LIN {X 0,Y 171.539,Z 336.57,A -85,B 0,C 180,E1 -22879.56,E2 -22879.56} C_VEL
LIN {X 0,Y 171.457,Z 336.598,A -85,B 0,C 180,E1 -22885.61,E2 -22885.61} C_VEL
LIN {X 0,Y 171.451,Z 336.623,A -85,B 0,C 180,E1 -22890.594,E2 -22890.594} C_VEL
LIN {X 0,Y 171.436,Z 336.681,A -85,B 0,C 180,E1 -22896.744,E2 -22896.744} C_VEL
LIN {X 0,Y 171.586,Z 337.511,A -85,B 0,C 180,E1 -22897.442,E2 -22897.442} C_VEL
LIN {X 0,Y 173.163,Z 340.46,A -85,B 0,C 180,E1 -22898.398,E2 -22898.398} C_VEL
LIN {X 0,Y 175.194,Z 342.365,A -85,B 0,C 180,E1 -22899.355,E2 -22899.355} C_VEL
LIN {X 0,Y 177.505,Z 345.855,A -85,B 0,C 180,E1 -22900.477,E2 -22900.477} C_VEL
LIN {X 0,Y 178.729,Z 347.281,A -85,B 0,C 180,E1 -22901.024,E2 -22901.024} C_VEL
LIN {X 0,Y 181.282,Z 350.846,A -85,B 0,C 180,E1 -22902.156,E2 -22902.156} C_VEL
LIN {X 0,Y 189.365,Z 363.13,A -85,B 0,C 180,E1 -22905.455,E2 -22905.455} C_VEL
LIN {X 0,Y 196.206,Z 374.838,A -85,B 0,C 180,E1 -22907.971,E2 -22907.971} C_VEL
LIN {X 0,Y 203.333,Z 389.329,A -85,B 0,C 180,E1 -22910.423,E2 -22910.423} C_VEL
LIN {X 0,Y 211.371,Z 406.535,A -85,B 0,C 180,E1 -22912.937,E2 -22912.937} C_VEL
LIN {X 0,Y 219.567,Z 420.322,A -85,B 0,C 180,E1 -22915.088,E2 -22915.088} C_VEL
LIN {X 0,Y 227.66,Z 431.79,A -85,B 0,C 180,E1 -22916.962,E2 -22916.962} C_VEL
LIN {X 0,Y 235.909,Z 442.056,A -85,B 0,C 180,E1 -22918.82,E2 -22918.82} C_VEL
LIN {X 0,Y 244.185,Z 451.427,A -85,B 0,C 180,E1 -22920.707,E2 -22920.707} C_VEL
LIN {X 0,Y 253.061,Z 460.521,A -85,B 0,C 180,E1 -22922.709,E2 -22922.709} C_VEL
LIN {X 0,Y 263.681,Z 469.922,A -85,B 0,C 180,E1 -22924.985,E2 -22924.985} C_VEL
LIN {X 0,Y 276.754,Z 479.974,A -85,B 0,C 180,E1 -22927.61,E2 -22927.61} C_VEL
LIN {X 0,Y 290.967,Z 490.138,A -85,B 0,C 180,E1 -22930.388,E2 -22930.388} C_VEL
LIN {X 0,Y 299.99,Z 496.755,A -85,B 0,C 180,E1 -22932.269,E2 -22932.269} C_VEL
LIN {X 0,Y 305.153,Z 500.286,A -85,B 0,C 180,E1 -22933.437,E2 -22933.437} C_VEL
LIN {X 0,Y 312.328,Z 505.427,A -85,B 0,C 180,E1 -22935.368,E2 -22935.368} C_VEL
LIN {X 0,Y 318.736,Z 509.419,A -85,B 0,C 180,E1 -22937.262,E2 -22937.262} C_VEL
LIN {X 0,Y 322.775,Z 512.115,A -85,B 0,C 180,E1 -22938.699,E2 -22938.699} C_VEL
LIN {X 0,Y 327.518,Z 515.418,A -85,B 0,C 180,E1 -22940.776,E2 -22940.776} C_VEL
LIN {X 0,Y 331.239,Z 517.603,A -85,B 0,C 180,E1 -22942.686,E2 -22942.686} C_VEL
LIN {X 0,Y 333.408,Z 518.666,A -85,B 0,C 180,E1 -22943.95,E2 -22943.95} C_VEL
LIN {X 0,Y 335.133,Z 519.458,A -85,B 0,C 180,E1 -22945.188,E2 -22945.188} C_VEL
LIN {X 0,Y 336.579,Z 519.977,A -85,B 0,C 180,E1 -22946.409,E2 -22946.409} C_VEL
LIN {X 0,Y 337.607,Z 520.419,A -85,B 0,C 180,E1 -22947.718,E2 -22947.718} C_VEL
LIN {X 0,Y 338.053,Z 520.65,A -85,B 0,C 180,E1 -22948.809,E2 -22948.809} C_VEL
LIN {X 0,Y 338.329,Z 520.665,A -85,B 0,C 180,E1 -22950,E2 -22950} C_VEL
LIN {X 0,Y 338.087,Z 520.616,A -85,B 0,C 180,E1 -22951.191,E2 -22951.191} C_VEL
LIN {X 0,Y 337.557,Z 520.347,A -85,B 0,C 180,E1 -22952.386,E2 -22952.386} C_VEL
LIN {X 0,Y 336.575,Z 519.955,A -85,B 0,C 180,E1 -22953.591,E2 -22953.591} C_VEL
LIN {X 0,Y 335.143,Z 519.423,A -85,B 0,C 180,E1 -22954.812,E2 -22954.812} C_VEL
LIN {X 0,Y 332.51,Z 518.272,A -85,B 0,C 180,E1 -22956.593,E2 -22956.593} C_VEL
LIN {X 0,Y 327.523,Z 515.378,A -85,B 0,C 180,E1 -22959.229,E2 -22959.229} C_VEL
LIN {X 0,Y 322.579,Z 512.01,A -85,B 0,C 180,E1 -22961.364,E2 -22961.364} C_VEL
LIN {X 0,Y 317.511,Z 508.69,A -85,B 0,C 180,E1 -22963.117,E2 -22963.117} C_VEL
LIN {X 0,Y 312.34,Z 505.397,A -85,B 0,C 180,E1 -22964.64,E2 -22964.64} C_VEL
LIN {X 0,Y 307.147,Z 501.743,A -85,B 0,C 180,E1 -22966.052,E2 -22966.052} C_VEL
LIN {X 0,Y 300.051,Z 496.781,A -85,B 0,C 180,E1 -22967.727,E2 -22967.727} C_VEL
LIN {X 0,Y 289.801,Z 489.324,A -85,B 0,C 180,E1 -22969.847,E2 -22969.847} C_VEL
LIN {X 0,Y 274.501,Z 478.341,A -85,B 0,C 180,E1 -22972.826,E2 -22972.826} C_VEL
LIN {X 0,Y 261.546,Z 468.134,A -85,B 0,C 180,E1 -22975.463,E2 -22975.463} C_VEL
LIN {X 0,Y 249.213,Z 456.773,A -85,B 0,C 180,E1 -22978.147,E2 -22978.147} C_VEL
LIN {X 0,Y 238.518,Z 445.13,A -85,B 0,C 180,E1 -22980.58,E2 -22980.58} C_VEL
LIN {X 0,Y 230.343,Z 435.166,A -85,B 0,C 180,E1 -22982.456,E2 -22982.456} C_VEL
LIN {X 0,Y 222.347,Z 424.476,A -85,B 0,C 180,E1 -22984.25,E2 -22984.25} C_VEL
LIN {X 0,Y 213.586,Z 410.542,A -85,B 0,C 180,E1 -22986.448,E2 -22986.448} C_VEL
LIN {X 0,Y 206.428,Z 396.381,A -85,B 0,C 180,E1 -22988.556,E2 -22988.556} C_VEL
LIN {X 0,Y 200.05,Z 382.426,A -85,B 0,C 180,E1 -22990.684,E2 -22990.684} C_VEL
LIN {X 0,Y 193.877,Z 370.717,A -85,B 0,C 180,E1 -22992.861,E2 -22992.861} C_VEL
LIN {X 0,Y 186.721,Z 358.92,A -85,B 0,C 180,E1 -22995.582,E2 -22995.582} C_VEL
LIN {X 0,Y 180.881,Z 350.422,A -85,B 0,C 180,E1 -22998.01,E2 -22998.01} C_VEL
LIN {X 0,Y 177.92,Z 346.242,A -85,B 0,C 180,E1 -22999.342,E2 -22999.342} C_VEL
LIN {X 0,Y 175.643,Z 343.253,A -85,B 0,C 180,E1 -23000.409,E2 -23000.409} C_VEL
LIN {X 0,Y 174.818,Z 341.844,A -85,B 0,C 180,E1 -23000.829,E2 -23000.829} C_VEL
LIN {X 0,Y 172.552,Z 339.652,A -85,B 0,C 180,E1 -23001.914,E2 -23001.914} C_VEL
LIN {X 0,Y 171.503,Z 337.185,A -85,B 0,C 180,E1 -23002.721,E2 -23002.721} C_VEL
LIN {X 0,Y 171.43,Z 336.639,A -85,B 0,C 180,E1 -23003.528,E2 -23003.528} C_VEL
LIN {X 0,Y 171.451,Z 336.623,A -85,B 0,C 180,E1 -23009.406,E2 -23009.406} C_VEL
LIN {X 0,Y 171.457,Z 336.598,A -85,B 0,C 180,E1 -23014.39,E2 -23014.39} C_VEL
LIN {X 0,Y 171.574,Z 336.565,A -85,B 0,C 180,E1 -23020.873,E2 -23020.873} C_VEL
LIN {X 0,Y 171.571,Z 336.612,A -85,B 0,C 180,E1 -23025.774,E2 -23025.774} C_VEL
LIN {X 0,Y 171.843,Z 336.526,A -85,B 0,C 180,E1 -23030.586,E2 -23030.586} C_VEL
LIN {X 0,Y 171.811,Z 336.582,A -85,B 0,C 180,E1 -23035.309,E2 -23035.309} C_VEL
LIN {X 0,Y 172.326,Z 336.463,A -85,B 0,C 180,E1 -23040.001,E2 -23040.001} C_VEL
LIN {X 0,Y 171.812,Z 336.584,A -85,B 0,C 180,E1 -23044.694,E2 -23044.694} C_VEL
LIN {X 0,Y 171.845,Z 336.523,A -85,B 0,C 180,E1 -23049.417,E2 -23049.417} C_VEL
LIN {X 0,Y 171.572,Z 336.611,A -85,B 0,C 180,E1 -23054.229,E2 -23054.229} C_VEL
LIN {X 0,Y 171.538,Z 336.57,A -85,B 0,C 180,E1 -23059.558,E2 -23059.558} C_VEL
LIN {X 0,Y 171.457,Z 336.59,A -85,B 0,C 180,E1 -23065.61,E2 -23065.61} C_VEL
LIN {X 0,Y 171.455,Z 336.629,A -85,B 0,C 180,E1 -23070.596,E2 -23070.596} C_VEL
LIN {X 0,Y 171.405,Z 336.708,A -85,B 0,C 180,E1 -23076.298,E2 -23076.298} C_VEL
LIN {X 0,Y 171.543,Z 337.483,A -85,B 0,C 180,E1 -23076.996,E2 -23076.996} C_VEL
LIN {X 0,Y 173.071,Z 340.36,A -85,B 0,C 180,E1 -23077.968,E2 -23077.968} C_VEL
LIN {X 0,Y 175.48,Z 343.334,A -85,B 0,C 180,E1 -23079.147,E2 -23079.147} C_VEL
LIN {X 0,Y 178.282,Z 347.76,A -85,B 0,C 180,E1 -23080.502,E2 -23080.502} C_VEL
LIN {X 0,Y 182.818,Z 355.351,A -85,B 0,C 180,E1 -23082.561,E2 -23082.561} C_VEL
LIN {X 0,Y 189.402,Z 367.454,A -85,B 0,C 180,E1 -23085.307,E2 -23085.307} C_VEL
LIN {X 0,Y 194.801,Z 378.934,A -85,B 0,C 180,E1 -23087.411,E2 -23087.411} C_VEL
LIN {X 0,Y 199.89,Z 391.574,A -85,B 0,C 180,E1 -23089.317,E2 -23089.317} C_VEL
LIN {X 0,Y 201.451,Z 403.372,A -85,B 0,C 180,E1 -23090.231,E2 -23090.231} C_VEL
LIN {X 0,Y 199.159,Z 444.488,A -85,B 0,C 180,E1 -23091.639,E2 -23091.639} C_VEL
LIN {X 0,Y 197.867,Z 455.855,A -85,B 0,C 180,E1 -23092.266,E2 -23092.266} C_VEL
LIN {X 0,Y 195.589,Z 468.974,A -85,B 0,C 180,E1 -23093.319,E2 -23093.319} C_VEL
LIN {X 0,Y 192.896,Z 480.518,A -85,B 0,C 180,E1 -23094.663,E2 -23094.663} C_VEL
LIN {X 0,Y 190.383,Z 489.79,A -85,B 0,C 180,E1 -23096.06,E2 -23096.06} C_VEL
LIN {X 0,Y 187.56,Z 498.728,A -85,B 0,C 180,E1 -23097.728,E2 -23097.728} C_VEL
LIN {X 0,Y 184.613,Z 507.253,A -85,B 0,C 180,E1 -23099.709,E2 -23099.709} C_VEL
LIN {X 0,Y 181.877,Z 514.468,A -85,B 0,C 180,E1 -23101.748,E2 -23101.748} C_VEL
LIN {X 0,Y 179.451,Z 520.668,A -85,B 0,C 180,E1 -23103.859,E2 -23103.859} C_VEL
LIN {X 0,Y 176.902,Z 527.209,A -85,B 0,C 180,E1 -23106.592,E2 -23106.592} C_VEL
LIN {X 0,Y 174.939,Z 531.708,A -85,B 0,C 180,E1 -23108.804,E2 -23108.804} C_VEL
LIN {X 0,Y 172.581,Z 537.2,A -85,B 0,C 180,E1 -23112.217,E2 -23112.217} C_VEL
LIN {X 0,Y 170.823,Z 541.528,A -85,B 0,C 180,E1 -23115.709,E2 -23115.709} C_VEL
LIN {X 0,Y 170.023,Z 543.9,A -85,B 0,C 180,E1 -23118.073,E2 -23118.073} C_VEL
LIN {X 0,Y 169.422,Z 545.703,A -85,B 0,C 180,E1 -23120.449,E2 -23120.449} C_VEL
LIN {X 0,Y 168.933,Z 548.162,A -85,B 0,C 180,E1 -23125.227,E2 -23125.227} C_VEL
LIN {X 0,Y 168.87,Z 548.808,A -85,B 0,C 180,E1 -23128.406,E2 -23128.406} C_VEL
LIN {X 0,Y 168.968,Z 548.914,A -85,B 0,C 180,E1 -23130,E2 -23130} C_VEL
LIN {X 0,Y 168.853,Z 548.695,A -85,B 0,C 180,E1 -23132.627,E2 -23132.627} C_VEL
LIN {X 0,Y 168.866,Z 548.16,A -85,B 0,C 180,E1 -23134.775,E2 -23134.775} C_VEL
LIN {X 0,Y 169.235,Z 546.252,A -85,B 0,C 180,E1 -23138.613,E2 -23138.613} C_VEL
LIN {X 0,Y 168.968,Z 544.98,A -85,B 0,C 180,E1 -23140.565,E2 -23140.565} C_VEL
LIN {X 0,Y 167.056,Z 542.347,A -85,B 0,C 180,E1 -23143.761,E2 -23143.761} C_VEL
LIN {X 0,Y 165.58,Z 539.031,A -85,B 0,C 180,E1 -23146.945,E2 -23146.945} C_VEL
LIN {X 0,Y 165.998,Z 536.621,A -85,B 0,C 180,E1 -23148.811,E2 -23148.811} C_VEL
LIN {X 0,Y 168.812,Z 530.478,A -85,B 0,C 180,E1 -23152.649,E2 -23152.649} C_VEL
LIN {X 0,Y 171.522,Z 524.246,A -85,B 0,C 180,E1 -23155.65,E2 -23155.65} C_VEL
LIN {X 0,Y 174.325,Z 517.526,A -85,B 0,C 180,E1 -23158.274,E2 -23158.274} C_VEL
LIN {X 0,Y 177.771,Z 508.977,A -85,B 0,C 180,E1 -23160.926,E2 -23160.926} C_VEL
LIN {X 0,Y 180.808,Z 500.803,A -85,B 0,C 180,E1 -23162.968,E2 -23162.968} C_VEL
LIN {X 0,Y 183.669,Z 492.297,A -85,B 0,C 180,E1 -23164.692,E2 -23164.692} C_VEL
LIN {X 0,Y 186.244,Z 483.585,A -85,B 0,C 180,E1 -23166.129,E2 -23166.129} C_VEL
LIN {X 0,Y 188.762,Z 473.833,A -85,B 0,C 180,E1 -23167.397,E2 -23167.397} C_VEL
LIN {X 0,Y 190.897,Z 463.758,A -85,B 0,C 180,E1 -23168.407,E2 -23168.407} C_VEL
LIN {X 0,Y 192.63,Z 453.291,A -85,B 0,C 180,E1 -23169.178,E2 -23169.178} C_VEL
LIN {X 0,Y 193.719,Z 443.215,A -85,B 0,C 180,E1 -23169.709,E2 -23169.709} C_VEL
LIN {X 0,Y 195.93,Z 403.202,A -85,B 0,C 180,E1 -23171.124,E2 -23171.124} C_VEL
LIN {X 0,Y 194.544,Z 393.897,A -85,B 0,C 180,E1 -23171.929,E2 -23171.929} C_VEL
LIN {X 0,Y 189.257,Z 380.763,A -85,B 0,C 180,E1 -23174.046,E2 -23174.046} C_VEL
LIN {X 0,Y 184.606,Z 370.872,A -85,B 0,C 180,E1 -23175.988,E2 -23175.988} C_VEL
LIN {X 0,Y 177.81,Z 358.124,A -85,B 0,C 180,E1 -23179.048,E2 -23179.048} C_VEL
LIN {X 0,Y 173.971,Z 351.983,A -85,B 0,C 180,E1 -23180.907,E2 -23180.907} C_VEL
LIN {X 0,Y 171.184,Z 347.548,A -85,B 0,C 180,E1 -23182.358,E2 -23182.358} C_VEL
LIN {X 0,Y 168.609,Z 344.054,A -85,B 0,C 180,E1 -23183.744,E2 -23183.744} C_VEL
LIN {X 0,Y 167.778,Z 342.747,A -85,B 0,C 180,E1 -23184.224,E2 -23184.224} C_VEL
LIN {X 0,Y 165.411,Z 340.457,A -85,B 0,C 180,E1 -23185.54,E2 -23185.54} C_VEL
LIN {X 0,Y 164.431,Z 338.113,A -85,B 0,C 180,E1 -23186.418,E2 -23186.418} C_VEL
LIN {X 0,Y 164.369,Z 337.528,A -85,B 0,C 180,E1 -23187.272,E2 -23187.272} C_VEL
LIN {X 0,Y 164.337,Z 337.477,A -85,B 0,C 180,E1 -23191.937,E2 -23191.937} C_VEL
LIN {X 0,Y 164.405,Z 337.47,A -85,B 0,C 180,E1 -23194.691,E2 -23194.691} C_VEL
LIN {X 0,Y 164.483,Z 337.45,A -85,B 0,C 180,E1 -23200.05,E2 -23200.05} C_VEL
LIN {X 0,Y 164.52,Z 337.482,A -85,B 0,C 180,E1 -23205.147,E2 -23205.147} C_VEL
LIN {X 0,Y 164.765,Z 337.405,A -85,B 0,C 180,E1 -23210.175,E2 -23210.175} C_VEL
LIN {X 0,Y 164.827,Z 337.411,A -85,B 0,C 180,E1 -23212.649,E2 -23212.649} C_VEL
LIN {X 0,Y 165.044,Z 337.393,A -85,B 0,C 180,E1 -23217.558,E2 -23217.558} C_VEL
LIN {X 0,Y 165.289,Z 337.339,A -85,B 0,C 180,E1 -23219.999,E2 -23219.999} C_VEL
LIN {X 0,Y 164.76,Z 337.461,A -85,B 0,C 180,E1 -23224.893,E2 -23224.893} C_VEL
LIN {X 0,Y 164.826,Z 337.421,A -85,B 0,C 180,E1 -23227.348,E2 -23227.348} C_VEL
LIN {X 0,Y 164.699,Z 337.418,A -85,B 0,C 180,E1 -23231.059,E2 -23231.059} C_VEL
LIN {X 0,Y 164.519,Z 337.493,A -85,B 0,C 180,E1 -23234.85,E2 -23234.85} C_VEL
LIN {X 0,Y 164.469,Z 337.452,A -85,B 0,C 180,E1 -23239.988,E2 -23239.988} C_VEL
LIN {X 0,Y 164.383,Z 337.474,A -85,B 0,C 180,E1 -23246.129,E2 -23246.129} C_VEL
LIN {X 0,Y 164.383,Z 337.492,A -85,B 0,C 180,E1 -23252.377,E2 -23252.377} C_VEL
LIN {X 0,Y 164.374,Z 337.825,A -85,B 0,C 180,E1 -23253.766,E2 -23253.766} C_VEL
LIN {X 0,Y 164.716,Z 339.072,A -85,B 0,C 180,E1 -23254.365,E2 -23254.365} C_VEL
LIN {X 0,Y 166.42,Z 341.678,A -85,B 0,C 180,E1 -23255.433,E2 -23255.433} C_VEL
LIN {X 0,Y 168.28,Z 343.196,A -85,B 0,C 180,E1 -23256.427,E2 -23256.427} C_VEL
LIN {X 0,Y 170.447,Z 346.622,A -85,B 0,C 180,E1 -23257.643,E2 -23257.643} C_VEL
LIN {X 0,Y 172.181,Z 348.499,A -85,B 0,C 180,E1 -23258.514,E2 -23258.514} C_VEL
LIN {X 0,Y 174.855,Z 352.169,A -85,B 0,C 180,E1 -23259.841,E2 -23259.841} C_VEL
LIN {X 0,Y 181.754,Z 362.408,A -85,B 0,C 180,E1 -23262.984,E2 -23262.984} C_VEL
LIN {X 0,Y 187.458,Z 371.661,A -85,B 0,C 180,E1 -23265.327,E2 -23265.327} C_VEL
LIN {X 0,Y 192.641,Z 380.983,A -85,B 0,C 180,E1 -23267.308,E2 -23267.308} C_VEL
LIN {X 0,Y 198.981,Z 394.263,A -85,B 0,C 180,E1 -23269.602,E2 -23269.602} C_VEL
LIN {X 0,Y 206.603,Z 410.847,A -85,B 0,C 180,E1 -23272.111,E2 -23272.111} C_VEL
LIN {X 0,Y 214.984,Z 425.115,A -85,B 0,C 180,E1 -23274.419,E2 -23274.419} C_VEL
LIN {X 0,Y 222.86,Z 436.51,A -85,B 0,C 180,E1 -23276.379,E2 -23276.379} C_VEL
LIN {X 0,Y 232.034,Z 448.156,A -85,B 0,C 180,E1 -23278.684,E2 -23278.684} C_VEL
LIN {X 0,Y 241.126,Z 458.487,A -85,B 0,C 180,E1 -23280.971,E2 -23280.971} C_VEL
LIN {X 0,Y 250.242,Z 467.531,A -85,B 0,C 180,E1 -23283.174,E2 -23283.174} C_VEL
LIN {X 0,Y 261.923,Z 477.462,A -85,B 0,C 180,E1 -23285.823,E2 -23285.823} C_VEL
LIN {X 0,Y 276.505,Z 488.237,A -85,B 0,C 180,E1 -23288.897,E2 -23288.897} C_VEL
LIN {X 0,Y 289.062,Z 496.933,A -85,B 0,C 180,E1 -23291.477,E2 -23291.477} C_VEL
LIN {X 0,Y 298.844,Z 503.742,A -85,B 0,C 180,E1 -23293.608,E2 -23293.608} C_VEL
LIN {X 0,Y 305.422,Z 508.49,A -85,B 0,C 180,E1 -23295.338,E2 -23295.338} C_VEL
LIN {X 0,Y 311.013,Z 512.125,A -85,B 0,C 180,E1 -23296.94,E2 -23296.94} C_VEL
LIN {X 0,Y 315.674,Z 515.006,A -85,B 0,C 180,E1 -23298.442,E2 -23298.442} C_VEL
LIN {X 0,Y 320.633,Z 518.493,A -85,B 0,C 180,E1 -23300.521,E2 -23300.521} C_VEL
LIN {X 0,Y 325.665,Z 521.536,A -85,B 0,C 180,E1 -23303.066,E2 -23303.066} C_VEL
LIN {X 0,Y 328.836,Z 523.081,A -85,B 0,C 180,E1 -23305.096,E2 -23305.096} C_VEL
LIN {X 0,Y 330.825,Z 523.835,A -85,B 0,C 180,E1 -23306.805,E2 -23306.805} C_VEL
LIN {X 0,Y 331.972,Z 524.341,A -85,B 0,C 180,E1 -23308.787,E2 -23308.787} C_VEL
LIN {X 0,Y 332.28,Z 524.36,A -85,B 0,C 180,E1 -23310,E2 -23310} C_VEL
LIN {X 0,Y 332.008,Z 524.312,A -85,B 0,C 180,E1 -23311.213,E2 -23311.213} C_VEL
LIN {X 0,Y 330.826,Z 523.842,A -85,B 0,C 180,E1 -23313.198,E2 -23313.198} C_VEL
LIN {X 0,Y 328.857,Z 523.049,A -85,B 0,C 180,E1 -23314.904,E2 -23314.904} C_VEL
LIN {X 0,Y 325.667,Z 521.523,A -85,B 0,C 180,E1 -23316.937,E2 -23316.937} C_VEL
LIN {X 0,Y 322.114,Z 519.453,A -85,B 0,C 180,E1 -23318.785,E2 -23318.785} C_VEL
LIN {X 0,Y 319.122,Z 517.476,A -85,B 0,C 180,E1 -23320.147,E2 -23320.147} C_VEL
LIN {X 0,Y 315.636,Z 515.014,A -85,B 0,C 180,E1 -23321.566,E2 -23321.566} C_VEL
LIN {X 0,Y 310.45,Z 511.729,A -85,B 0,C 180,E1 -23323.239,E2 -23323.239} C_VEL
LIN {X 0,Y 305.201,Z 508.34,A -85,B 0,C 180,E1 -23324.729,E2 -23324.729} C_VEL
LIN {X 0,Y 298.749,Z 503.734,A -85,B 0,C 180,E1 -23326.397,E2 -23326.397} C_VEL
LIN {X 0,Y 291.782,Z 498.874,A -85,B 0,C 180,E1 -23327.939,E2 -23327.939} C_VEL
LIN {X 0,Y 283.585,Z 493.015,A -85,B 0,C 180,E1 -23329.656,E2 -23329.656} C_VEL
LIN {X 0,Y 272.673,Z 485.406,A -85,B 0,C 180,E1 -23331.896,E2 -23331.896} C_VEL
LIN {X 0,Y 261.917,Z 477.484,A -85,B 0,C 180,E1 -23334.175,E2 -23334.175} C_VEL
LIN {X 0,Y 250.239,Z 467.543,A -85,B 0,C 180,E1 -23336.824,E2 -23336.824} C_VEL
LIN {X 0,Y 241.128,Z 458.477,A -85,B 0,C 180,E1 -23339.029,E2 -23339.029} C_VEL
LIN {X 0,Y 230.977,Z 446.931,A -85,B 0,C 180,E1 -23341.576,E2 -23341.576} C_VEL
LIN {X 0,Y 221.582,Z 434.806,A -85,B 0,C 180,E1 -23343.944,E2 -23343.944} C_VEL
LIN {X 0,Y 211.908,Z 420.264,A -85,B 0,C 180,E1 -23346.383,E2 -23346.383} C_VEL
LIN {X 0,Y 204.622,Z 406.869,A -85,B 0,C 180,E1 -23348.5,E2 -23348.5} C_VEL
LIN {X 0,Y 195.301,Z 386.39,A -85,B 0,C 180,E1 -23351.709,E2 -23351.709} C_VEL
LIN {X 0,Y 189.403,Z 374.942,A -85,B 0,C 180,E1 -23353.92,E2 -23353.92} C_VEL
LIN {X 0,Y 182.781,Z 363.899,A -85,B 0,C 180,E1 -23356.585,E2 -23356.585} C_VEL
LIN {X 0,Y 176.957,Z 355.329,A -85,B 0,C 180,E1 -23359.151,E2 -23359.151} C_VEL
LIN {X 0,Y 174.25,Z 351.474,A -85,B 0,C 180,E1 -23360.444,E2 -23360.444} C_VEL
LIN {X 0,Y 171.46,Z 347.586,A -85,B 0,C 180,E1 -23361.853,E2 -23361.853} C_VEL
LIN {X 0,Y 169.045,Z 344.703,A -85,B 0,C 180,E1 -23363.115,E2 -23363.115} C_VEL
LIN {X 0,Y 167.929,Z 342.817,A -85,B 0,C 180,E1 -23363.763,E2 -23363.763} C_VEL
LIN {X 0,Y 165.707,Z 340.823,A -85,B 0,C 180,E1 -23364.981,E2 -23364.981} C_VEL
LIN {X 0,Y 164.437,Z 338.037,A -85,B 0,C 180,E1 -23366.04,E2 -23366.04} C_VEL
LIN {X 0,Y 164.342,Z 337.513,A -85,B 0,C 180,E1 -23366.923,E2 -23366.923} C_VEL
LIN {X 0,Y 164.398,Z 337.505,A -85,B 0,C 180,E1 -23369.138,E2 -23369.138} C_VEL
LIN {X 0,Y 164.405,Z 337.479,A -85,B 0,C 180,E1 -23374.694,E2 -23374.694} C_VEL
LIN {X 0,Y 164.481,Z 337.45,A -85,B 0,C 180,E1 -23380.052,E2 -23380.052} C_VEL
LIN {X 0,Y 164.519,Z 337.493,A -85,B 0,C 180,E1 -23385.15,E2 -23385.15} C_VEL
LIN {X 0,Y 164.763,Z 337.407,A -85,B 0,C 180,E1 -23390.178,E2 -23390.178} C_VEL
LIN {X 0,Y 164.826,Z 337.421,A -85,B 0,C 180,E1 -23392.652,E2 -23392.652} C_VEL
LIN {X 0,Y 165.043,Z 337.383,A -85,B 0,C 180,E1 -23397.561,E2 -23397.561} C_VEL
LIN {X 0,Y 165.289,Z 337.339,A -85,B 0,C 180,E1 -23400.001,E2 -23400.001} C_VEL
LIN {X 0,Y 164.761,Z 337.461,A -85,B 0,C 180,E1 -23404.895,E2 -23404.895} C_VEL
LIN {X 0,Y 164.827,Z 337.411,A -85,B 0,C 180,E1 -23407.351,E2 -23407.351} C_VEL
LIN {X 0,Y 164.7,Z 337.42,A -85,B 0,C 180,E1 -23411.062,E2 -23411.062} C_VEL
LIN {X 0,Y 164.478,Z 337.449,A -85,B 0,C 180,E1 -23417.405,E2 -23417.405} C_VEL
LIN {X 0,Y 164.471,Z 337.452,A -85,B 0,C 180,E1 -23419.991,E2 -23419.991} C_VEL
LIN {X 0,Y 164.384,Z 337.468,A -85,B 0,C 180,E1 -23426.129,E2 -23426.129} C_VEL
LIN {X 0,Y 164.385,Z 337.5,A -85,B 0,C 180,E1 -23432.38,E2 -23432.38} C_VEL
LIN {X 0,Y 164.408,Z 337.879,A -85,B 0,C 180,E1 -23433.413,E2 -23433.413} C_VEL
LIN {X 0,Y 164.788,Z 339.234,A -85,B 0,C 180,E1 -23434.036,E2 -23434.036} C_VEL
LIN {X 0,Y 166.493,Z 341.748,A -85,B 0,C 180,E1 -23435.089,E2 -23435.089} C_VEL
LIN {X 0,Y 168.296,Z 343.276,A -85,B 0,C 180,E1 -23436.056,E2 -23436.056} C_VEL
LIN {X 0,Y 170.346,Z 346.513,A -85,B 0,C 180,E1 -23437.207,E2 -23437.207} C_VEL
LIN {X 0,Y 172.227,Z 349.051,A -85,B 0,C 180,E1 -23438.185,E2 -23438.185} C_VEL
LIN {X 0,Y 176.235,Z 355.622,A -85,B 0,C 180,E1 -23440.209,E2 -23440.209} C_VEL
LIN {X 0,Y 180.315,Z 362.639,A -85,B 0,C 180,E1 -23442.117,E2 -23442.117} C_VEL
LIN {X 0,Y 187.188,Z 376.123,A -85,B 0,C 180,E1 -23445.097,E2 -23445.097} C_VEL
LIN {X 0,Y 192.937,Z 389.661,A -85,B 0,C 180,E1 -23447.435,E2 -23447.435} C_VEL
LIN {X 0,Y 194.8,Z 394.774,A -85,B 0,C 180,E1 -23448.181,E2 -23448.181} C_VEL
LIN {X 0,Y 195.977,Z 403.646,A -85,B 0,C 180,E1 -23448.909,E2 -23448.909} C_VEL
LIN {X 0,Y 193.648,Z 444.156,A -85,B 0,C 180,E1 -23450.327,E2 -23450.327} C_VEL
LIN {X 0,Y 192.398,Z 454.945,A -85,B 0,C 180,E1 -23450.925,E2 -23450.925} C_VEL
LIN {X 0,Y 190.447,Z 466.333,A -85,B 0,C 180,E1 -23451.822,E2 -23451.822} C_VEL
LIN {X 0,Y 187.641,Z 478.692,A -85,B 0,C 180,E1 -23453.183,E2 -23453.183} C_VEL
LIN {X 0,Y 184.536,Z 489.596,A -85,B 0,C 180,E1 -23454.829,E2 -23454.829} C_VEL
LIN {X 0,Y 181.597,Z 498.534,A -85,B 0,C 180,E1 -23456.532,E2 -23456.532} C_VEL
LIN {X 0,Y 178.487,Z 507.058,A -85,B 0,C 180,E1 -23458.553,E2 -23458.553} C_VEL
LIN {X 0,Y 175.632,Z 514.273,A -85,B 0,C 180,E1 -23460.648,E2 -23460.648} C_VEL
LIN {X 0,Y 173.076,Z 520.473,A -85,B 0,C 180,E1 -23462.818,E2 -23462.818} C_VEL
LIN {X 0,Y 170.38,Z 527.014,A -85,B 0,C 180,E1 -23465.639,E2 -23465.639} C_VEL
LIN {X 0,Y 168.309,Z 531.513,A -85,B 0,C 180,E1 -23467.926,E2 -23467.926} C_VEL
LIN {X 0,Y 165.822,Z 537.006,A -85,B 0,C 180,E1 -23471.466,E2 -23471.466} C_VEL
LIN {X 0,Y 163.901,Z 541.333,A -85,B 0,C 180,E1 -23475.092,E2 -23475.092} C_VEL
LIN {X 0,Y 163.054,Z 543.705,A -85,B 0,C 180,E1 -23477.555,E2 -23477.555} C_VEL
LIN {X 0,Y 162.403,Z 545.509,A -85,B 0,C 180,E1 -23480.032,E2 -23480.032} C_VEL
LIN {X 0,Y 161.852,Z 547.968,A -85,B 0,C 180,E1 -23485.018,E2 -23485.018} C_VEL
LIN {X 0,Y 161.8,Z 548.562,A -85,B 0,C 180,E1 -23487.511,E2 -23487.511} C_VEL
LIN {X 0,Y 161.884,Z 548.721,A -85,B 0,C 180,E1 -23490,E2 -23490} C_VEL
LIN {X 0,Y 161.763,Z 548.561,A -85,B 0,C 180,E1 -23492.49,E2 -23492.49} C_VEL
LIN {X 0,Y 161.771,Z 547.966,A -85,B 0,C 180,E1 -23494.984,E2 -23494.984} C_VEL
LIN {X 0,Y 162.4,Z 545.509,A -85,B 0,C 180,E1 -23499.968,E2 -23499.968} C_VEL
LIN {X 0,Y 163.453,Z 542.552,A -85,B 0,C 180,E1 -23503.679,E2 -23503.679} C_VEL
LIN {X 0,Y 165.066,Z 538.559,A -85,B 0,C 180,E1 -23507.339,E2 -23507.339} C_VEL
LIN {X 0,Y 165.998,Z 536.621,A -85,B 0,C 180,E1 -23508.811,E2 -23508.811} C_VEL
LIN {X 0,Y 166.559,Z 534.024,A -85,B 0,C 180,E1 -23510.629,E2 -23510.629} C_VEL
LIN {X 0,Y 165.964,Z 529.362,A -85,B 0,C 180,E1 -23513.643,E2 -23513.643} C_VEL
LIN {X 0,Y 165.65,Z 524.205,A -85,B 0,C 180,E1 -23516.563,E2 -23516.563} C_VEL
LIN {X 0,Y 166.625,Z 520.588,A -85,B 0,C 180,E1 -23518.173,E2 -23518.173} C_VEL
LIN {X 0,Y 170.198,Z 512.453,A -85,B 0,C 180,E1 -23521.074,E2 -23521.074} C_VEL
LIN {X 0,Y 174.459,Z 501.742,A -85,B 0,C 180,E1 -23523.982,E2 -23523.982} C_VEL
LIN {X 0,Y 177.461,Z 493.455,A -85,B 0,C 180,E1 -23525.742,E2 -23525.742} C_VEL
LIN {X 0,Y 180.554,Z 483.391,A -85,B 0,C 180,E1 -23527.458,E2 -23527.458} C_VEL
LIN {X 0,Y 183.181,Z 473.64,A -85,B 0,C 180,E1 -23528.744,E2 -23528.744} C_VEL
LIN {X 0,Y 185.391,Z 463.564,A -85,B 0,C 180,E1 -23529.769,E2 -23529.769} C_VEL
LIN {X 0,Y 187.175,Z 453.147,A -85,B 0,C 180,E1 -23530.547,E2 -23530.547} C_VEL
LIN {X 0,Y 188.292,Z 443.238,A -85,B 0,C 180,E1 -23531.08,E2 -23531.08} C_VEL
LIN {X 0,Y 190.573,Z 404.451,A -85,B 0,C 180,E1 -23532.474,E2 -23532.474} C_VEL
LIN {X 0,Y 189.457,Z 396.777,A -85,B 0,C 180,E1 -23533.17,E2 -23533.17} C_VEL
LIN {X 0,Y 184.427,Z 384.044,A -85,B 0,C 180,E1 -23535.328,E2 -23535.328} C_VEL
LIN {X 0,Y 180.286,Z 375.137,A -85,B 0,C 180,E1 -23537.173,E2 -23537.173} C_VEL
LIN {X 0,Y 174.016,Z 363.082,A -85,B 0,C 180,E1 -23540.186,E2 -23540.186} C_VEL
LIN {X 0,Y 170.397,Z 357.048,A -85,B 0,C 180,E1 -23542.061,E2 -23542.061} C_VEL
LIN {X 0,Y 167.74,Z 352.846,A -85,B 0,C 180,E1 -23543.526,E2 -23543.526} C_VEL
LIN {X 0,Y 164.723,Z 348.661,A -85,B 0,C 180,E1 -23545.271,E2 -23545.271} C_VEL
LIN {X 0,Y 162.165,Z 345.621,A -85,B 0,C 180,E1 -23546.827,E2 -23546.827} C_VEL
LIN {X 0,Y 161.152,Z 343.832,A -85,B 0,C 180,E1 -23547.522,E2 -23547.522} C_VEL
LIN {X 0,Y 158.719,Z 341.761,A -85,B 0,C 180,E1 -23549.095,E2 -23549.095} C_VEL
LIN {X 0,Y 157.402,Z 338.94,A -85,B 0,C 180,E1 -23550.399,E2 -23550.399} C_VEL
LIN {X 0,Y 157.293,Z 338.412,A -85,B 0,C 180,E1 -23551.293,E2 -23551.293} C_VEL
LIN {X 0,Y 157.302,Z 338.376,A -85,B 0,C 180,E1 -23556.289,E2 -23556.289} C_VEL
LIN {X 0,Y 157.406,Z 338.325,A -85,B 0,C 180,E1 -23561.786,E2 -23561.786} C_VEL
LIN {X 0,Y 157.526,Z 338.34,A -85,B 0,C 180,E1 -23567.109,E2 -23567.109} C_VEL
LIN {X 0,Y 157.686,Z 338.287,A -85,B 0,C 180,E1 -23569.729,E2 -23569.729} C_VEL
LIN {X 0,Y 157.764,Z 338.285,A -85,B 0,C 180,E1 -23572.318,E2 -23572.318} C_VEL
LIN {X 0,Y 158.252,Z 338.215,A -85,B 0,C 180,E1 -23579.999,E2 -23579.999} C_VEL
LIN {X 0,Y 157.763,Z 338.294,A -85,B 0,C 180,E1 -23587.679,E2 -23587.679} C_VEL
LIN {X 0,Y 157.63,Z 338.299,A -85,B 0,C 180,E1 -23591.229,E2 -23591.229} C_VEL
LIN {X 0,Y 157.449,Z 338.363,A -85,B 0,C 180,E1 -23595.533,E2 -23595.533} C_VEL
LIN {X 0,Y 157.365,Z 338.343,A -85,B 0,C 180,E1 -23600.932,E2 -23600.932} C_VEL
LIN {X 0,Y 157.305,Z 338.351,A -85,B 0,C 180,E1 -23606.68,E2 -23606.68} C_VEL
LIN {X 0,Y 157.336,Z 338.675,A -85,B 0,C 180,E1 -23609.704,E2 -23609.704} C_VEL
LIN {X 0,Y 157.686,Z 339.847,A -85,B 0,C 180,E1 -23610.461,E2 -23610.461} C_VEL
LIN {X 0,Y 159.21,Z 342.375,A -85,B 0,C 180,E1 -23611.633,E2 -23611.633} C_VEL
LIN {X 0,Y 161.456,Z 344.136,A -85,B 0,C 180,E1 -23613.055,E2 -23613.055} C_VEL
LIN {X 0,Y 163.488,Z 347.447,A -85,B 0,C 180,E1 -23614.395,E2 -23614.395} C_VEL
LIN {X 0,Y 165.523,Z 349.552,A -85,B 0,C 180,E1 -23615.573,E2 -23615.573} C_VEL
LIN {X 0,Y 168.088,Z 353.12,A -85,B 0,C 180,E1 -23617.036,E2 -23617.036} C_VEL
LIN {X 0,Y 169.381,Z 354.84,A -85,B 0,C 180,E1 -23617.733,E2 -23617.733} C_VEL
LIN {X 0,Y 172.835,Z 359.785,A -85,B 0,C 180,E1 -23619.518,E2 -23619.518} C_VEL
LIN {X 0,Y 177.448,Z 366.628,A -85,B 0,C 180,E1 -23621.713,E2 -23621.713} C_VEL
LIN {X 0,Y 183.213,Z 376.139,A -85,B 0,C 180,E1 -23624.238,E2 -23624.238} C_VEL
LIN {X 0,Y 188.806,Z 386.509,A -85,B 0,C 180,E1 -23626.503,E2 -23626.503} C_VEL
LIN {X 0,Y 194.884,Z 399.727,A -85,B 0,C 180,E1 -23628.826,E2 -23628.826} C_VEL
LIN {X 0,Y 201.868,Z 415.137,A -85,B 0,C 180,E1 -23631.243,E2 -23631.243} C_VEL
LIN {X 0,Y 210.208,Z 429.561,A -85,B 0,C 180,E1 -23633.66,E2 -23633.66} C_VEL
LIN {X 0,Y 217.978,Z 441.2,A -85,B 0,C 180,E1 -23635.811,E2 -23635.811} C_VEL
LIN {X 0,Y 226.168,Z 451.966,A -85,B 0,C 180,E1 -23638.113,E2 -23638.113} C_VEL
LIN {X 0,Y 235.644,Z 462.961,A -85,B 0,C 180,E1 -23640.733,E2 -23640.733} C_VEL
LIN {X 0,Y 244.421,Z 471.804,A -85,B 0,C 180,E1 -23643.043,E2 -23643.043} C_VEL
LIN {X 0,Y 254.732,Z 480.684,A -85,B 0,C 180,E1 -23645.567,E2 -23645.567} C_VEL
LIN {X 0,Y 269.065,Z 491.142,A -85,B 0,C 180,E1 -23648.784,E2 -23648.784} C_VEL
LIN {X 0,Y 281.649,Z 499.573,A -85,B 0,C 180,E1 -23651.478,E2 -23651.478} C_VEL
LIN {X 0,Y 292.58,Z 506.972,A -85,B 0,C 180,E1 -23653.907,E2 -23653.907} C_VEL
LIN {X 0,Y 299.526,Z 511.961,A -85,B 0,C 180,E1 -23655.705,E2 -23655.705} C_VEL
LIN {X 0,Y 304.711,Z 515.359,A -85,B 0,C 180,E1 -23657.169,E2 -23657.169} C_VEL
LIN {X 0,Y 309.779,Z 518.479,A -85,B 0,C 180,E1 -23658.776,E2 -23658.776} C_VEL
LIN {X 0,Y 313.638,Z 521.233,A -85,B 0,C 180,E1 -23660.38,E2 -23660.38} C_VEL
LIN {X 0,Y 318.729,Z 524.435,A -85,B 0,C 180,E1 -23662.857,E2 -23662.857} C_VEL
LIN {X 0,Y 322.203,Z 526.16,A -85,B 0,C 180,E1 -23664.995,E2 -23664.995} C_VEL
LIN {X 0,Y 323.942,Z 526.888,A -85,B 0,C 180,E1 -23666.345,E2 -23666.345} C_VEL
LIN {X 0,Y 325.024,Z 527.31,A -85,B 0,C 180,E1 -23667.521,E2 -23667.521} C_VEL
LIN {X 0,Y 325.649,Z 527.595,A -85,B 0,C 180,E1 -23668.763,E2 -23668.763} C_VEL
LIN {X 0,Y 325.969,Z 527.628,A -85,B 0,C 180,E1 -23670,E2 -23670} C_VEL
LIN {X 0,Y 325.678,Z 527.574,A -85,B 0,C 180,E1 -23671.236,E2 -23671.236} C_VEL
LIN {X 0,Y 325.06,Z 527.283,A -85,B 0,C 180,E1 -23672.478,E2 -23672.478} C_VEL
LIN {X 0,Y 323.852,Z 526.836,A -85,B 0,C 180,E1 -23673.733,E2 -23673.733} C_VEL
LIN {X 0,Y 322.21,Z 526.152,A -85,B 0,C 180,E1 -23675.005,E2 -23675.005} C_VEL
LIN {X 0,Y 318.726,Z 524.412,A -85,B 0,C 180,E1 -23677.139,E2 -23677.139} C_VEL
LIN {X 0,Y 315.043,Z 522.188,A -85,B 0,C 180,E1 -23678.984,E2 -23678.984} C_VEL
LIN {X 0,Y 311.837,Z 519.993,A -85,B 0,C 180,E1 -23680.387,E2 -23680.387} C_VEL
LIN {X 0,Y 307.879,Z 517.302,A -85,B 0,C 180,E1 -23681.855,E2 -23681.855} C_VEL
LIN {X 0,Y 302.663,Z 514.008,A -85,B 0,C 180,E1 -23683.427,E2 -23683.427} C_VEL
LIN {X 0,Y 296.485,Z 509.768,A -85,B 0,C 180,E1 -23685.114,E2 -23685.114} C_VEL
LIN {X 0,Y 289.832,Z 505.13,A -85,B 0,C 180,E1 -23686.707,E2 -23686.707} C_VEL
LIN {X 0,Y 278.891,Z 497.712,A -85,B 0,C 180,E1 -23689.123,E2 -23689.123} C_VEL
LIN {X 0,Y 263.55,Z 487.305,A -85,B 0,C 180,E1 -23692.421,E2 -23692.421} C_VEL
LIN {X 0,Y 249.539,Z 476.427,A -85,B 0,C 180,E1 -23695.68,E2 -23695.68} C_VEL
LIN {X 0,Y 238.129,Z 465.627,A -85,B 0,C 180,E1 -23698.597,E2 -23698.597} C_VEL
LIN {X 0,Y 229.474,Z 455.989,A -85,B 0,C 180,E1 -23700.96,E2 -23700.96} C_VEL
LIN {X 0,Y 221.812,Z 446.367,A -85,B 0,C 180,E1 -23703.108,E2 -23703.108} C_VEL
LIN {X 0,Y 214.424,Z 436.075,A -85,B 0,C 180,E1 -23705.181,E2 -23705.181} C_VEL
LIN {X 0,Y 205.815,Z 422.308,A -85,B 0,C 180,E1 -23707.564,E2 -23707.564} C_VEL
LIN {X 0,Y 198.397,Z 407.975,A -85,B 0,C 180,E1 -23709.903,E2 -23709.903} C_VEL
LIN {X 0,Y 191.357,Z 391.852,A -85,B 0,C 180,E1 -23712.504,E2 -23712.504} C_VEL
LIN {X 0,Y 185.215,Z 379.634,A -85,B 0,C 180,E1 -23714.936,E2 -23714.936} C_VEL
LIN {X 0,Y 178.88,Z 368.878,A -85,B 0,C 180,E1 -23717.639,E2 -23717.639} C_VEL
LIN {X 0,Y 173.049,Z 360.07,A -85,B 0,C 180,E1 -23720.378,E2 -23720.378} C_VEL
LIN {X 0,Y 170.441,Z 356.41,A -85,B 0,C 180,E1 -23721.7,E2 -23721.7} C_VEL
LIN {X 0,Y 168.09,Z 353.097,A -85,B 0,C 180,E1 -23722.964,E2 -23722.964} C_VEL
LIN {X 0,Y 165.617,Z 349.712,A -85,B 0,C 180,E1 -23724.369,E2 -23724.369} C_VEL
LIN {X 0,Y 164.51,Z 348.481,A -85,B 0,C 180,E1 -23725.007,E2 -23725.007} C_VEL
LIN {X 0,Y 162.152,Z 345.545,A -85,B 0,C 180,E1 -23726.455,E2 -23726.455} C_VEL
LIN {X 0,Y 161.133,Z 343.819,A -85,B 0,C 180,E1 -23727.149,E2 -23727.149} C_VEL
LIN {X 0,Y 158.72,Z 341.794,A -85,B 0,C 180,E1 -23728.708,E2 -23728.708} C_VEL
LIN {X 0,Y 157.459,Z 339.135,A -85,B 0,C 180,E1 -23729.861,E2 -23729.861} C_VEL
LIN {X 0,Y 157.277,Z 338.435,A -85,B 0,C 180,E1 -23730.927,E2 -23730.927} C_VEL
LIN {X 0,Y 157.311,Z 338.351,A -85,B 0,C 180,E1 -23733.466,E2 -23733.466} C_VEL
LIN {X 0,Y 157.389,Z 338.335,A -85,B 0,C 180,E1 -23739.669,E2 -23739.669} C_VEL
LIN {X 0,Y 157.449,Z 338.363,A -85,B 0,C 180,E1 -23744.467,E2 -23744.467} C_VEL
LIN {X 0,Y 157.685,Z 338.288,A -85,B 0,C 180,E1 -23749.732,E2 -23749.732} C_VEL
LIN {X 0,Y 157.763,Z 338.294,A -85,B 0,C 180,E1 -23752.321,E2 -23752.321} C_VEL
LIN {X 0,Y 158.252,Z 338.215,A -85,B 0,C 180,E1 -23760.001,E2 -23760.001} C_VEL
LIN {X 0,Y 157.764,Z 338.285,A -85,B 0,C 180,E1 -23767.682,E2 -23767.682} C_VEL
LIN {X 0,Y 157.634,Z 338.301,A -85,B 0,C 180,E1 -23771.237,E2 -23771.237} C_VEL
LIN {X 0,Y 157.449,Z 338.347,A -85,B 0,C 180,E1 -23775.536,E2 -23775.536} C_VEL
LIN {X 0,Y 157.366,Z 338.347,A -85,B 0,C 180,E1 -23780.935,E2 -23780.935} C_VEL
LIN {X 0,Y 157.309,Z 338.347,A -85,B 0,C 180,E1 -23786.682,E2 -23786.682} C_VEL
LIN {X 0,Y 157.332,Z 338.688,A -85,B 0,C 180,E1 -23789.34,E2 -23789.34} C_VEL
LIN {X 0,Y 157.694,Z 339.93,A -85,B 0,C 180,E1 -23790.093,E2 -23790.093} C_VEL
LIN {X 0,Y 159.354,Z 342.471,A -85,B 0,C 180,E1 -23791.341,E2 -23791.341} C_VEL
LIN {X 0,Y 161.469,Z 344.22,A -85,B 0,C 180,E1 -23792.684,E2 -23792.684} C_VEL
LIN {X 0,Y 163.446,Z 347.415,A -85,B 0,C 180,E1 -23793.987,E2 -23793.987} C_VEL
LIN {X 0,Y 165.486,Z 349.56,A -85,B 0,C 180,E1 -23795.172,E2 -23795.172} C_VEL
LIN {X 0,Y 168.9,Z 354.484,A -85,B 0,C 180,E1 -23797.112,E2 -23797.112} C_VEL
LIN {X 0,Y 172.833,Z 361.129,A -85,B 0,C 180,E1 -23799.219,E2 -23799.219} C_VEL
LIN {X 0,Y 176.747,Z 368.169,A -85,B 0,C 180,E1 -23801.165,E2 -23801.165} C_VEL
LIN {X 0,Y 183.046,Z 380.837,A -85,B 0,C 180,E1 -23804.059,E2 -23804.059} C_VEL
LIN {X 0,Y 188.232,Z 393.47,A -85,B 0,C 180,E1 -23806.312,E2 -23806.312} C_VEL
LIN {X 0,Y 189.743,Z 397.833,A -85,B 0,C 180,E1 -23806.964,E2 -23806.964} C_VEL
LIN {X 0,Y 190.614,Z 404.876,A -85,B 0,C 180,E1 -23807.558,E2 -23807.558} C_VEL
LIN {X 0,Y 188.224,Z 443.969,A -85,B 0,C 180,E1 -23808.943,E2 -23808.943} C_VEL
LIN {X 0,Y 186.952,Z 454.69,A -85,B 0,C 180,E1 -23809.551,E2 -23809.551} C_VEL
LIN {X 0,Y 184.929,Z 466.14,A -85,B 0,C 180,E1 -23810.465,E2 -23810.465} C_VEL
LIN {X 0,Y 181.994,Z 478.498,A -85,B 0,C 180,E1 -23811.841,E2 -23811.841} C_VEL
LIN {X 0,Y 178.775,Z 489.402,A -85,B 0,C 180,E1 -23813.517,E2 -23813.517} C_VEL
LIN {X 0,Y 175.707,Z 498.34,A -85,B 0,C 180,E1 -23815.252,E2 -23815.252} C_VEL
LIN {X 0,Y 172.439,Z 506.863,A -85,B 0,C 180,E1 -23817.316,E2 -23817.316} C_VEL
LIN {X 0,Y 169.467,Z 514.079,A -85,B 0,C 180,E1 -23819.469,E2 -23819.469} C_VEL
LIN {X 0,Y 166.759,Z 520.279,A -85,B 0,C 180,E1 -23821.698,E2 -23821.698} C_VEL
LIN {X 0,Y 164.625,Z 525.053,A -85,B 0,C 180,E1 -23823.706,E2 -23823.706} C_VEL
LIN {X 0,Y 161.734,Z 531.319,A -85,B 0,C 180,E1 -23826.978,E2 -23826.978} C_VEL
LIN {X 0,Y 159.07,Z 536.811,A -85,B 0,C 180,E1 -23830.649,E2 -23830.649} C_VEL
LIN {X 0,Y 157.004,Z 541.137,A -85,B 0,C 180,E1 -23834.421,E2 -23834.421} C_VEL
LIN {X 0,Y 156.083,Z 543.51,A -85,B 0,C 180,E1 -23836.989,E2 -23836.989} C_VEL
LIN {X 0,Y 155.404,Z 545.315,A -85,B 0,C 180,E1 -23839.578,E2 -23839.578} C_VEL
LIN {X 0,Y 154.754,Z 547.773,A -85,B 0,C 180,E1 -23844.789,E2 -23844.789} C_VEL
LIN {X 0,Y 154.715,Z 548.489,A -85,B 0,C 180,E1 -23847.983,E2 -23847.983} C_VEL
LIN {X 0,Y 154.687,Z 548.519,A -85,B 0,C 180,E1 -23851.695,E2 -23851.695} C_VEL
LIN {X 0,Y 154.698,Z 547.772,A -85,B 0,C 180,E1 -23855.213,E2 -23855.213} C_VEL
LIN {X 0,Y 155.402,Z 545.315,A -85,B 0,C 180,E1 -23860.422,E2 -23860.422} C_VEL
LIN {X 0,Y 156.527,Z 542.357,A -85,B 0,C 180,E1 -23864.297,E2 -23864.297} C_VEL
LIN {X 0,Y 158.291,Z 538.365,A -85,B 0,C 180,E1 -23868.107,E2 -23868.107} C_VEL
LIN {X 0,Y 160.784,Z 533.235,A -85,B 0,C 180,E1 -23871.81,E2 -23871.81} C_VEL
LIN {X 0,Y 163.376,Z 527.975,A -85,B 0,C 180,E1 -23874.797,E2 -23874.797} C_VEL
LIN {X 0,Y 165.496,Z 523.181,A -85,B 0,C 180,E1 -23877.087,E2 -23877.087} C_VEL
LIN {X 0,Y 166.625,Z 520.588,A -85,B 0,C 180,E1 -23878.173,E2 -23878.173} C_VEL
LIN {X 0,Y 167.687,Z 516.899,A -85,B 0,C 180,E1 -23879.713,E2 -23879.713} C_VEL
LIN {X 0,Y 167.945,Z 510.491,A -85,B 0,C 180,E1 -23882.302,E2 -23882.302} C_VEL
LIN {X 0,Y 168.386,Z 503.603,A -85,B 0,C 180,E1 -23884.721,E2 -23884.721} C_VEL
LIN {X 0,Y 169.598,Z 499.013,A -85,B 0,C 180,E1 -23885.912,E2 -23885.912} C_VEL
LIN {X 0,Y 172.624,Z 490.558,A -85,B 0,C 180,E1 -23887.639,E2 -23887.639} C_VEL
LIN {X 0,Y 175.431,Z 481.566,A -85,B 0,C 180,E1 -23889.12,E2 -23889.12} C_VEL
LIN {X 0,Y 178.182,Z 471.432,A -85,B 0,C 180,E1 -23890.416,E2 -23890.416} C_VEL
LIN {X 0,Y 180.479,Z 460.795,A -85,B 0,C 180,E1 -23891.451,E2 -23891.451} C_VEL
LIN {X 0,Y 182.629,Z 447.153,A -85,B 0,C 180,E1 -23892.36,E2 -23892.36} C_VEL
LIN {X 0,Y 184.04,Z 427.854,A -85,B 0,C 180,E1 -23893.118,E2 -23893.118} C_VEL
LIN {X 0,Y 185.345,Z 405.488,A -85,B 0,C 180,E1 -23893.907,E2 -23893.907} C_VEL
LIN {X 0,Y 184.461,Z 399.538,A -85,B 0,C 180,E1 -23894.486,E2 -23894.486} C_VEL
LIN {X 0,Y 178.852,Z 385.304,A -85,B 0,C 180,E1 -23897.08,E2 -23897.08} C_VEL
LIN {X 0,Y 173.523,Z 374.233,A -85,B 0,C 180,E1 -23899.68,E2 -23899.68} C_VEL
LIN {X 0,Y 169.24,Z 366.196,A -85,B 0,C 180,E1 -23901.944,E2 -23901.944} C_VEL
LIN {X 0,Y 164.997,Z 358.907,A -85,B 0,C 180,E1 -23904.381,E2 -23904.381} C_VEL
LIN {X 0,Y 161.744,Z 354.471,A -85,B 0,C 180,E1 -23906.356,E2 -23906.356} C_VEL
LIN {X 0,Y 159.121,Z 350.983,A -85,B 0,C 180,E1 -23908.081,E2 -23908.081} C_VEL
LIN {X 0,Y 158.292,Z 349.886,A -85,B 0,C 180,E1 -23908.655,E2 -23908.655} C_VEL
LIN {X 0,Y 155.885,Z 347.318,A -85,B 0,C 180,E1 -23910.36,E2 -23910.36} C_VEL
LIN {X 0,Y 154.529,Z 344.939,A -85,B 0,C 180,E1 -23911.473,E2 -23911.473} C_VEL
LIN {X 0,Y 151.893,Z 342.943,A -85,B 0,C 180,E1 -23913.55,E2 -23913.55} C_VEL
LIN {X 0,Y 150.461,Z 340.398,A -85,B 0,C 180,E1 -23915.007,E2 -23915.007} C_VEL
LIN {X 0,Y 150.27,Z 339.503,A -85,B 0,C 180,E1 -23915.842,E2 -23915.842} C_VEL
LIN {X 0,Y 150.337,Z 339.206,A -85,B 0,C 180,E1 -23920.897,E2 -23920.897} C_VEL
LIN {X 0,Y 150.433,Z 339.234,A -85,B 0,C 180,E1 -23926.49,E2 -23926.49} C_VEL
LIN {X 0,Y 150.608,Z 339.171,A -85,B 0,C 180,E1 -23929.241,E2 -23929.241} C_VEL
LIN {X 0,Y 150.686,Z 339.162,A -85,B 0,C 180,E1 -23931.955,E2 -23931.955} C_VEL
LIN {X 0,Y 151.212,Z 339.091,A -85,B 0,C 180,E1 -23939.999,E2 -23939.999} C_VEL
LIN {X 0,Y 150.684,Z 339.169,A -85,B 0,C 180,E1 -23948.042,E2 -23948.042} C_VEL
LIN {X 0,Y 150.571,Z 339.179,A -85,B 0,C 180,E1 -23951.431,E2 -23951.431} C_VEL
LIN {X 0,Y 150.356,Z 339.23,A -85,B 0,C 180,E1 -23956.286,E2 -23956.286} C_VEL
LIN {X 0,Y 150.347,Z 339.215,A -85,B 0,C 180,E1 -23960.791,E2 -23960.791} C_VEL
LIN {X 0,Y 150.259,Z 339.503,A -85,B 0,C 180,E1 -23964.616,E2 -23964.616} C_VEL
LIN {X 0,Y 150.546,Z 340.644,A -85,B 0,C 180,E1 -23965.503,E2 -23965.503} C_VEL
LIN {X 0,Y 152.18,Z 343.245,A -85,B 0,C 180,E1 -23967.08,E2 -23967.08} C_VEL
LIN {X 0,Y 154.885,Z 345.404,A -85,B 0,C 180,E1 -23969.194,E2 -23969.194} C_VEL
LIN {X 0,Y 156.758,Z 348.503,A -85,B 0,C 180,E1 -23970.681,E2 -23970.681} C_VEL
LIN {X 0,Y 158.913,Z 350.55,A -85,B 0,C 180,E1 -23972.148,E2 -23972.148} C_VEL
LIN {X 0,Y 161.396,Z 354.127,A -85,B 0,C 180,E1 -23973.816,E2 -23973.816} C_VEL
LIN {X 0,Y 162.839,Z 355.787,A -85,B 0,C 180,E1 -23974.699,E2 -23974.699} C_VEL
LIN {X 0,Y 166.647,Z 361.105,A -85,B 0,C 180,E1 -23976.937,E2 -23976.937} C_VEL
LIN {X 0,Y 171.297,Z 367.832,A -85,B 0,C 180,E1 -23979.411,E2 -23979.411} C_VEL
LIN {X 0,Y 177.741,Z 378.303,A -85,B 0,C 180,E1 -23982.511,E2 -23982.511} C_VEL
LIN {X 0,Y 183.745,Z 389.44,A -85,B 0,C 180,E1 -23985.135,E2 -23985.135} C_VEL
LIN {X 0,Y 189.627,Z 402.356,A -85,B 0,C 180,E1 -23987.544,E2 -23987.544} C_VEL
LIN {X 0,Y 197.118,Z 419.299,A -85,B 0,C 180,E1 -23990.312,E2 -23990.312} C_VEL
LIN {X 0,Y 204.945,Z 433.277,A -85,B 0,C 180,E1 -23992.769,E2 -23992.769} C_VEL
LIN {X 0,Y 211.513,Z 443.677,A -85,B 0,C 180,E1 -23994.802,E2 -23994.802} C_VEL
LIN {X 0,Y 218.171,Z 452.982,A -85,B 0,C 180,E1 -23996.88,E2 -23996.88} C_VEL
LIN {X 0,Y 226.071,Z 462.829,A -85,B 0,C 180,E1 -23999.31,E2 -23999.31} C_VEL
LIN {X 0,Y 234.954,Z 472.545,A -85,B 0,C 180,E1 -24001.932,E2 -24001.932} C_VEL
LIN {X 0,Y 246.242,Z 482.778,A -85,B 0,C 180,E1 -24004.979,E2 -24004.979} C_VEL
LIN {X 0,Y 257.981,Z 491.611,A -85,B 0,C 180,E1 -24007.853,E2 -24007.853} C_VEL
LIN {X 0,Y 271.462,Z 500.529,A -85,B 0,C 180,E1 -24010.899,E2 -24010.899} C_VEL
LIN {X 0,Y 282.381,Z 507.521,A -85,B 0,C 180,E1 -24013.373,E2 -24013.373} C_VEL
LIN {X 0,Y 287.867,Z 511.019,A -85,B 0,C 180,E1 -24014.65,E2 -24014.65} C_VEL
LIN {X 0,Y 293.534,Z 515.006,A -85,B 0,C 180,E1 -24016.148,E2 -24016.148} C_VEL
LIN {X 0,Y 299.406,Z 518.869,A -85,B 0,C 180,E1 -24017.804,E2 -24017.804} C_VEL
LIN {X 0,Y 304.137,Z 521.83,A -85,B 0,C 180,E1 -24019.347,E2 -24019.347} C_VEL
LIN {X 0,Y 307.638,Z 524.273,A -85,B 0,C 180,E1 -24020.798,E2 -24020.798} C_VEL
LIN {X 0,Y 311.707,Z 526.848,A -85,B 0,C 180,E1 -24022.768,E2 -24022.768} C_VEL
LIN {X 0,Y 315.289,Z 528.772,A -85,B 0,C 180,E1 -24024.885,E2 -24024.885} C_VEL
LIN {X 0,Y 317.053,Z 529.514,A -85,B 0,C 180,E1 -24026.187,E2 -24026.187} C_VEL
LIN {X 0,Y 318.367,Z 530.015,A -85,B 0,C 180,E1 -24027.47,E2 -24027.47} C_VEL
LIN {X 0,Y 319.082,Z 530.335,A -85,B 0,C 180,E1 -24028.738,E2 -24028.738} C_VEL
LIN {X 0,Y 319.445,Z 530.393,A -85,B 0,C 180,E1 -24030,E2 -24030} C_VEL
LIN {X 0,Y 319.107,Z 530.322,A -85,B 0,C 180,E1 -24031.262,E2 -24031.262} C_VEL
LIN {X 0,Y 318.391,Z 530.004,A -85,B 0,C 180,E1 -24032.53,E2 -24032.53} C_VEL
LIN {X 0,Y 316.981,Z 529.486,A -85,B 0,C 180,E1 -24033.878,E2 -24033.878} C_VEL
LIN {X 0,Y 315.297,Z 528.771,A -85,B 0,C 180,E1 -24035.115,E2 -24035.115} C_VEL
LIN {X 0,Y 311.707,Z 526.837,A -85,B 0,C 180,E1 -24037.232,E2 -24037.232} C_VEL
LIN {X 0,Y 307.604,Z 524.263,A -85,B 0,C 180,E1 -24039.203,E2 -24039.203} C_VEL
LIN {X 0,Y 304.105,Z 521.824,A -85,B 0,C 180,E1 -24040.654,E2 -24040.654} C_VEL
LIN {X 0,Y 298.293,Z 518.15,A -85,B 0,C 180,E1 -24042.54,E2 -24042.54} C_VEL
LIN {X 0,Y 290.565,Z 512.906,A -85,B 0,C 180,E1 -24044.652,E2 -24044.652} C_VEL
LIN {X 0,Y 282.382,Z 507.516,A -85,B 0,C 180,E1 -24046.628,E2 -24046.628} C_VEL
LIN {X 0,Y 271.46,Z 500.538,A -85,B 0,C 180,E1 -24049.099,E2 -24049.099} C_VEL
LIN {X 0,Y 257.99,Z 491.584,A -85,B 0,C 180,E1 -24052.152,E2 -24052.152} C_VEL
LIN {X 0,Y 244.967,Z 481.688,A -85,B 0,C 180,E1 -24055.353,E2 -24055.353} C_VEL
LIN {X 0,Y 234.955,Z 472.541,A -85,B 0,C 180,E1 -24058.068,E2 -24058.068} C_VEL
LIN {X 0,Y 226.049,Z 462.851,A -85,B 0,C 180,E1 -24060.69,E2 -24060.69} C_VEL
LIN {X 0,Y 217.126,Z 451.551,A -85,B 0,C 180,E1 -24063.459,E2 -24063.459} C_VEL
LIN {X 0,Y 209.028,Z 439.814,A -85,B 0,C 180,E1 -24066,E2 -24066} C_VEL
LIN {X 0,Y 201.34,Z 427.118,A -85,B 0,C 180,E1 -24068.342,E2 -24068.342} C_VEL
LIN {X 0,Y 193.858,Z 412.463,A -85,B 0,C 180,E1 -24070.826,E2 -24070.826} C_VEL
LIN {X 0,Y 186.813,Z 396.019,A -85,B 0,C 180,E1 -24073.585,E2 -24073.585} C_VEL
LIN {X 0,Y 181.374,Z 384.826,A -85,B 0,C 180,E1 -24075.877,E2 -24075.877} C_VEL
LIN {X 0,Y 175.222,Z 374.085,A -85,B 0,C 180,E1 -24078.659,E2 -24078.659} C_VEL
LIN {X 0,Y 169.467,Z 365.122,A -85,B 0,C 180,E1 -24081.534,E2 -24081.534} C_VEL
LIN {X 0,Y 165.082,Z 358.897,A -85,B 0,C 180,E1 -24083.957,E2 -24083.957} C_VEL
LIN {X 0,Y 161.952,Z 354.669,A -85,B 0,C 180,E1 -24085.847,E2 -24085.847} C_VEL
LIN {X 0,Y 159.311,Z 351.278,A -85,B 0,C 180,E1 -24087.563,E2 -24087.563} C_VEL
LIN {X 0,Y 158.417,Z 349.969,A -85,B 0,C 180,E1 -24088.19,E2 -24088.19} C_VEL
LIN {X 0,Y 156.017,Z 347.531,A -85,B 0,C 180,E1 -24089.872,E2 -24089.872} C_VEL
LIN {X 0,Y 154.509,Z 344.952,A -85,B 0,C 180,E1 -24091.101,E2 -24091.101} C_VEL
LIN {X 0,Y 151.778,Z 342.809,A -85,B 0,C 180,E1 -24093.266,E2 -24093.266} C_VEL
LIN {X 0,Y 150.366,Z 340.009,A -85,B 0,C 180,E1 -24094.861,E2 -24094.861} C_VEL
LIN {X 0,Y 150.258,Z 339.303,A -85,B 0,C 180,E1 -24096.21,E2 -24096.21} C_VEL
LIN {X 0,Y 150.336,Z 339.209,A -85,B 0,C 180,E1 -24100.9,E2 -24100.9} C_VEL
LIN {X 0,Y 150.425,Z 339.226,A -85,B 0,C 180,E1 -24106.492,E2 -24106.492} C_VEL
LIN {X 0,Y 150.605,Z 339.17,A -85,B 0,C 180,E1 -24109.244,E2 -24109.244} C_VEL
LIN {X 0,Y 150.684,Z 339.169,A -85,B 0,C 180,E1 -24111.958,E2 -24111.958} C_VEL
LIN {X 0,Y 151.212,Z 339.091,A -85,B 0,C 180,E1 -24120.001,E2 -24120.001} C_VEL
LIN {X 0,Y 150.686,Z 339.162,A -85,B 0,C 180,E1 -24128.045,E2 -24128.045} C_VEL
LIN {X 0,Y 150.575,Z 339.181,A -85,B 0,C 180,E1 -24131.438,E2 -24131.438} C_VEL
LIN {X 0,Y 150.357,Z 339.217,A -85,B 0,C 180,E1 -24136.289,E2 -24136.289} C_VEL
LIN {X 0,Y 150.348,Z 339.218,A -85,B 0,C 180,E1 -24140.792,E2 -24140.792} C_VEL
LIN {X 0,Y 150.279,Z 339.536,A -85,B 0,C 180,E1 -24144.248,E2 -24144.248} C_VEL
LIN {X 0,Y 150.591,Z 340.727,A -85,B 0,C 180,E1 -24145.168,E2 -24145.168} C_VEL
LIN {X 0,Y 152.022,Z 343.052,A -85,B 0,C 180,E1 -24146.558,E2 -24146.558} C_VEL
LIN {X 0,Y 154.81,Z 345.28,A -85,B 0,C 180,E1 -24148.748,E2 -24148.748} C_VEL
LIN {X 0,Y 156.718,Z 348.44,A -85,B 0,C 180,E1 -24150.266,E2 -24150.266} C_VEL
LIN {X 0,Y 158.943,Z 350.583,A -85,B 0,C 180,E1 -24151.783,E2 -24151.783} C_VEL
LIN {X 0,Y 161.302,Z 354.024,A -85,B 0,C 180,E1 -24153.374,E2 -24153.374} C_VEL
LIN {X 0,Y 162.836,Z 355.823,A -85,B 0,C 180,E1 -24154.316,E2 -24154.316} C_VEL
LIN {X 0,Y 165.772,Z 360.201,A -85,B 0,C 180,E1 -24156.081,E2 -24156.081} C_VEL
LIN {X 0,Y 170.66,Z 368.569,A -85,B 0,C 180,E1 -24158.812,E2 -24158.812} C_VEL
LIN {X 0,Y 177.54,Z 382.417,A -85,B 0,C 180,E1 -24162.297,E2 -24162.297} C_VEL
LIN {X 0,Y 182.809,Z 395.072,A -85,B 0,C 180,E1 -24164.764,E2 -24164.764} C_VEL
LIN {X 0,Y 184.819,Z 400.979,A -85,B 0,C 180,E1 -24165.699,E2 -24165.699} C_VEL
LIN {X 0,Y 185.361,Z 406.526,A -85,B 0,C 180,E1 -24166.152,E2 -24166.152} C_VEL
LIN {X 0,Y 182.928,Z 443.653,A -85,B 0,C 180,E1 -24167.473,E2 -24167.473} C_VEL
LIN {X 0,Y 181.679,Z 454.025,A -85,B 0,C 180,E1 -24168.067,E2 -24168.067} C_VEL
LIN {X 0,Y 179.791,Z 464.659,A -85,B 0,C 180,E1 -24168.915,E2 -24168.915} C_VEL
LIN {X 0,Y 177.196,Z 475.459,A -85,B 0,C 180,E1 -24170.058,E2 -24170.058} C_VEL
LIN {X 0,Y 173.565,Z 487.856,A -85,B 0,C 180,E1 -24171.867,E2 -24171.867} C_VEL
LIN {X 0,Y 169.918,Z 498.146,A -85,B 0,C 180,E1 -24173.887,E2 -24173.887} C_VEL
LIN {X 0,Y 166.499,Z 506.669,A -85,B 0,C 180,E1 -24175.994,E2 -24175.994} C_VEL
LIN {X 0,Y 163.365,Z 513.884,A -85,B 0,C 180,E1 -24178.198,E2 -24178.198} C_VEL
LIN {X 0,Y 160.511,Z 520.084,A -85,B 0,C 180,E1 -24180.49,E2 -24180.49} C_VEL
LIN {X 0,Y 157.441,Z 526.623,A -85,B 0,C 180,E1 -24183.488,E2 -24183.488} C_VEL
LIN {X 0,Y 155.214,Z 531.125,A -85,B 0,C 180,E1 -24185.952,E2 -24185.952} C_VEL
LIN {X 0,Y 152.362,Z 536.616,A -85,B 0,C 180,E1 -24189.761,E2 -24189.761} C_VEL
LIN {X 0,Y 150.136,Z 540.942,A -85,B 0,C 180,E1 -24193.689,E2 -24193.689} C_VEL
LIN {X 0,Y 149.138,Z 543.315,A -85,B 0,C 180,E1 -24196.372,E2 -24196.372} C_VEL
LIN {X 0,Y 148.391,Z 545.12,A -85,B 0,C 180,E1 -24199.08,E2 -24199.08} C_VEL
LIN {X 0,Y 147.686,Z 547.58,A -85,B 0,C 180,E1 -24204.539,E2 -24204.539} C_VEL
LIN {X 0,Y 147.628,Z 548.331,A -85,B 0,C 180,E1 -24208.73,E2 -24208.73} C_VEL
LIN {X 0,Y 147.571,Z 548.173,A -85,B 0,C 180,E1 -24212.73,E2 -24212.73} C_VEL
LIN {X 0,Y 147.625,Z 547.578,A -85,B 0,C 180,E1 -24215.464,E2 -24215.464} C_VEL
LIN {X 0,Y 148.389,Z 545.12,A -85,B 0,C 180,E1 -24220.92,E2 -24220.92} C_VEL
LIN {X 0,Y 149.626,Z 542.163,A -85,B 0,C 180,E1 -24224.971,E2 -24224.971} C_VEL
LIN {X 0,Y 151.546,Z 538.17,A -85,B 0,C 180,E1 -24228.942,E2 -24228.942} C_VEL
LIN {X 0,Y 154.172,Z 533.04,A -85,B 0,C 180,E1 -24232.797,E2 -24232.797} C_VEL
LIN {X 0,Y 156.925,Z 527.78,A -85,B 0,C 180,E1 -24235.89,E2 -24235.89} C_VEL
LIN {X 0,Y 159.244,Z 522.799,A -85,B 0,C 180,E1 -24238.341,E2 -24238.341} C_VEL
LIN {X 0,Y 161.902,Z 517.137,A -85,B 0,C 180,E1 -24240.667,E2 -24240.667} C_VEL
LIN {X 0,Y 165.72,Z 508.588,A -85,B 0,C 180,E1 -24243.456,E2 -24243.456} C_VEL
LIN {X 0,Y 169.059,Z 500.414,A -85,B 0,C 180,E1 -24245.59,E2 -24245.59} C_VEL
LIN {X 0,Y 169.598,Z 499.013,A -85,B 0,C 180,E1 -24245.912,E2 -24245.912} C_VEL
LIN {X 0,Y 170.232,Z 495.961,A -85,B 0,C 180,E1 -24246.736,E2 -24246.736} C_VEL
LIN {X 0,Y 169.085,Z 485.977,A -85,B 0,C 180,E1 -24249.792,E2 -24249.792} C_VEL
LIN {X 0,Y 169.634,Z 482.507,A -85,B 0,C 180,E1 -24250.459,E2 -24250.459} C_VEL
LIN {X 0,Y 172.332,Z 473.252,A -85,B 0,C 180,E1 -24251.7,E2 -24251.7} C_VEL
LIN {X 0,Y 174.718,Z 463.176,A -85,B 0,C 180,E1 -24252.748,E2 -24252.748} C_VEL
LIN {X 0,Y 176.508,Z 453.522,A -85,B 0,C 180,E1 -24253.494,E2 -24253.494} C_VEL
LIN {X 0,Y 177.813,Z 443.106,A -85,B 0,C 180,E1 -24254.075,E2 -24254.075} C_VEL
LIN {X 0,Y 180.225,Z 406.695,A -85,B 0,C 180,E1 -24255.417,E2 -24255.417} C_VEL
LIN {X 0,Y 179.578,Z 402.497,A -85,B 0,C 180,E1 -24255.86,E2 -24255.86} C_VEL
LIN {X 0,Y 174.313,Z 388.725,A -85,B 0,C 180,E1 -24258.49,E2 -24258.49} C_VEL
LIN {X 0,Y 168.306,Z 376.111,A -85,B 0,C 180,E1 -24261.678,E2 -24261.678} C_VEL
LIN {X 0,Y 163.873,Z 367.922,A -85,B 0,C 180,E1 -24264.265,E2 -24264.265} C_VEL
LIN {X 0,Y 161.496,Z 363.97,A -85,B 0,C 180,E1 -24265.749,E2 -24265.749} C_VEL
LIN {X 0,Y 158.794,Z 360.164,A -85,B 0,C 180,E1 -24267.508,E2 -24267.508} C_VEL
LIN {X 0,Y 155.898,Z 356.178,A -85,B 0,C 180,E1 -24269.558,E2 -24269.558} C_VEL
LIN {X 0,Y 153.282,Z 353.073,A -85,B 0,C 180,E1 -24271.547,E2 -24271.547} C_VEL
LIN {X 0,Y 152.179,Z 351.298,A -85,B 0,C 180,E1 -24272.493,E2 -24272.493} C_VEL
LIN {X 0,Y 149.57,Z 348.969,A -85,B 0,C 180,E1 -24274.715,E2 -24274.715} C_VEL
LIN {X 0,Y 147.818,Z 345.969,A -85,B 0,C 180,E1 -24276.533,E2 -24276.533} C_VEL
LIN {X 0,Y 145.215,Z 344.124,A -85,B 0,C 180,E1 -24279.248,E2 -24279.248} C_VEL
LIN {X 0,Y 143.603,Z 341.496,A -85,B 0,C 180,E1 -24281.45,E2 -24281.45} C_VEL
LIN {X 0,Y 143.329,Z 340.377,A -85,B 0,C 180,E1 -24282.797,E2 -24282.797} C_VEL
LIN {X 0,Y 143.534,Z 340.055,A -85,B 0,C 180,E1 -24288.704,E2 -24288.704} C_VEL
LIN {X 0,Y 143.61,Z 340.04,A -85,B 0,C 180,E1 -24291.556,E2 -24291.556} C_VEL
LIN {X 0,Y 144.171,Z 339.967,A -85,B 0,C 180,E1 -24299.998,E2 -24299.998} C_VEL
LIN {X 0,Y 143.609,Z 340.046,A -85,B 0,C 180,E1 -24308.441,E2 -24308.441} C_VEL
LIN {X 0,Y 143.498,Z 340.06,A -85,B 0,C 180,E1 -24311.622,E2 -24311.622} C_VEL
LIN {X 0,Y 143.31,Z 340.37,A -85,B 0,C 180,E1 -24317.57,E2 -24317.57} C_VEL
LIN {X 0,Y 143.599,Z 341.447,A -85,B 0,C 180,E1 -24318.918,E2 -24318.918} C_VEL
LIN {X 0,Y 145.182,Z 344.127,A -85,B 0,C 180,E1 -24321.103,E2 -24321.103} C_VEL
LIN {X 0,Y 147.805,Z 345.95,A -85,B 0,C 180,E1 -24323.837,E2 -24323.837} C_VEL
LIN {X 0,Y 150.187,Z 349.69,A -85,B 0,C 180,E1 -24326.235,E2 -24326.235} C_VEL
LIN {X 0,Y 152.619,Z 351.833,A -85,B 0,C 180,E1 -24328.256,E2 -24328.256} C_VEL
LIN {X 0,Y 154.717,Z 355.055,A -85,B 0,C 180,E1 -24329.977,E2 -24329.977} C_VEL
LIN {X 0,Y 156.537,Z 357.011,A -85,B 0,C 180,E1 -24331.292,E2 -24331.292} C_VEL
LIN {X 0,Y 159.385,Z 360.803,A -85,B 0,C 180,E1 -24333.257,E2 -24333.257} C_VEL
LIN {X 0,Y 163.664,Z 366.891,A -85,B 0,C 180,E1 -24335.942,E2 -24335.942} C_VEL
LIN {X 0,Y 167.982,Z 373.349,A -85,B 0,C 180,E1 -24338.38,E2 -24338.38} C_VEL
LIN {X 0,Y 173.963,Z 383.323,A -85,B 0,C 180,E1 -24341.434,E2 -24341.434} C_VEL
LIN {X 0,Y 179.608,Z 394.09,A -85,B 0,C 180,E1 -24344.06,E2 -24344.06} C_VEL
LIN {X 0,Y 185.238,Z 406.863,A -85,B 0,C 180,E1 -24346.518,E2 -24346.518} C_VEL
LIN {X 0,Y 191.977,Z 422.511,A -85,B 0,C 180,E1 -24349.173,E2 -24349.173} C_VEL
LIN {X 0,Y 199.43,Z 436.474,A -85,B 0,C 180,E1 -24351.737,E2 -24351.737} C_VEL
LIN {X 0,Y 206.276,Z 447.868,A -85,B 0,C 180,E1 -24354.118,E2 -24354.118} C_VEL
LIN {X 0,Y 214.467,Z 459.536,A -85,B 0,C 180,E1 -24356.961,E2 -24356.961} C_VEL
LIN {X 0,Y 223.309,Z 470.428,A -85,B 0,C 180,E1 -24359.934,E2 -24359.934} C_VEL
LIN {X 0,Y 232.85,Z 480.359,A -85,B 0,C 180,E1 -24362.921,E2 -24362.921} C_VEL
LIN {X 0,Y 242.85,Z 488.854,A -85,B 0,C 180,E1 -24365.729,E2 -24365.729} C_VEL
LIN {X 0,Y 256.353,Z 498.364,A -85,B 0,C 180,E1 -24369.121,E2 -24369.121} C_VEL
LIN {X 0,Y 269.439,Z 506.468,A -85,B 0,C 180,E1 -24372.181,E2 -24372.181} C_VEL
LIN {X 0,Y 280.409,Z 513.11,A -85,B 0,C 180,E1 -24374.78,E2 -24374.78} C_VEL
LIN {X 0,Y 285.856,Z 516.628,A -85,B 0,C 180,E1 -24376.194,E2 -24376.194} C_VEL
LIN {X 0,Y 291.621,Z 520.412,A -85,B 0,C 180,E1 -24377.799,E2 -24377.799} C_VEL
LIN {X 0,Y 298.011,Z 524.455,A -85,B 0,C 180,E1 -24379.813,E2 -24379.813} C_VEL
LIN {X 0,Y 303.022,Z 527.873,A -85,B 0,C 180,E1 -24382.001,E2 -24382.001} C_VEL
LIN {X 0,Y 305.818,Z 529.555,A -85,B 0,C 180,E1 -24383.402,E2 -24383.402} C_VEL
LIN {X 0,Y 308.113,Z 530.783,A -85,B 0,C 180,E1 -24384.765,E2 -24384.765} C_VEL
LIN {X 0,Y 310.054,Z 531.684,A -85,B 0,C 180,E1 -24386.101,E2 -24386.101} C_VEL
LIN {X 0,Y 311.475,Z 532.244,A -85,B 0,C 180,E1 -24387.414,E2 -24387.414} C_VEL
LIN {X 0,Y 312.301,Z 532.574,A -85,B 0,C 180,E1 -24388.711,E2 -24388.711} C_VEL
LIN {X 0,Y 312.714,Z 532.643,A -85,B 0,C 180,E1 -24390,E2 -24390} C_VEL
LIN {X 0,Y 312.352,Z 532.561,A -85,B 0,C 180,E1 -24391.289,E2 -24391.289} C_VEL
LIN {X 0,Y 311.512,Z 532.237,A -85,B 0,C 180,E1 -24392.586,E2 -24392.586} C_VEL
LIN {X 0,Y 309.969,Z 531.657,A -85,B 0,C 180,E1 -24393.966,E2 -24393.966} C_VEL
LIN {X 0,Y 308.139,Z 530.796,A -85,B 0,C 180,E1 -24395.234,E2 -24395.234} C_VEL
LIN {X 0,Y 304.62,Z 528.851,A -85,B 0,C 180,E1 -24397.228,E2 -24397.228} C_VEL
LIN {X 0,Y 299.807,Z 525.669,A -85,B 0,C 180,E1 -24399.444,E2 -24399.444} C_VEL
LIN {X 0,Y 297.98,Z 524.457,A -85,B 0,C 180,E1 -24400.188,E2 -24400.188} C_VEL
LIN {X 0,Y 294.04,Z 521.888,A -85,B 0,C 180,E1 -24401.494,E2 -24401.494} C_VEL
LIN {X 0,Y 288.574,Z 518.422,A -85,B 0,C 180,E1 -24403.055,E2 -24403.055} C_VEL
LIN {X 0,Y 283.138,Z 514.857,A -85,B 0,C 180,E1 -24404.526,E2 -24404.526} C_VEL
LIN {X 0,Y 273.825,Z 509.201,A -85,B 0,C 180,E1 -24406.771,E2 -24406.771} C_VEL
LIN {X 0,Y 263.682,Z 503.042,A -85,B 0,C 180,E1 -24409.134,E2 -24409.134} C_VEL
LIN {X 0,Y 252.333,Z 495.731,A -85,B 0,C 180,E1 -24411.84,E2 -24411.84} C_VEL
LIN {X 0,Y 240.303,Z 486.805,A -85,B 0,C 180,E1 -24414.958,E2 -24414.958} C_VEL
LIN {X 0,Y 229.541,Z 477.112,A -85,B 0,C 180,E1 -24418.094,E2 -24418.094} C_VEL
LIN {X 0,Y 219.809,Z 466.369,A -85,B 0,C 180,E1 -24421.211,E2 -24421.211} C_VEL
LIN {X 0,Y 213.123,Z 457.792,A -85,B 0,C 180,E1 -24423.49,E2 -24423.49} C_VEL
LIN {X 0,Y 205.704,Z 446.949,A -85,B 0,C 180,E1 -24426.079,E2 -24426.079} C_VEL
LIN {X 0,Y 198.598,Z 434.988,A -85,B 0,C 180,E1 -24428.571,E2 -24428.571} C_VEL
LIN {X 0,Y 191.06,Z 420.578,A -85,B 0,C 180,E1 -24431.161,E2 -24431.161} C_VEL
LIN {X 0,Y 181.848,Z 398.985,A -85,B 0,C 180,E1 -24434.941,E2 -24434.941} C_VEL
LIN {X 0,Y 176.571,Z 388.102,A -85,B 0,C 180,E1 -24437.327,E2 -24437.327} C_VEL
LIN {X 0,Y 171.106,Z 378.442,A -85,B 0,C 180,E1 -24439.981,E2 -24439.981} C_VEL
LIN {X 0,Y 165.069,Z 368.837,A -85,B 0,C 180,E1 -24443.246,E2 -24443.246} C_VEL
LIN {X 0,Y 161.964,Z 364.463,A -85,B 0,C 180,E1 -24445.086,E2 -24445.086} C_VEL
LIN {X 0,Y 159.06,Z 360.478,A -85,B 0,C 180,E1 -24446.949,E2 -24446.949} C_VEL
LIN {X 0,Y 156.328,Z 356.63,A -85,B 0,C 180,E1 -24448.869,E2 -24448.869} C_VEL
LIN {X 0,Y 153.31,Z 353.167,A -85,B 0,C 180,E1 -24451.135,E2 -24451.135} C_VEL
LIN {X 0,Y 152.35,Z 351.463,A -85,B 0,C 180,E1 -24451.97,E2 -24451.97} C_VEL
LIN {X 0,Y 149.583,Z 348.968,A -85,B 0,C 180,E1 -24454.321,E2 -24454.321} C_VEL
LIN {X 0,Y 147.803,Z 345.969,A -85,B 0,C 180,E1 -24456.162,E2 -24456.162} C_VEL
LIN {X 0,Y 145.183,Z 344.115,A -85,B 0,C 180,E1 -24458.897,E2 -24458.897} C_VEL
LIN {X 0,Y 143.517,Z 341.234,A -85,B 0,C 180,E1 -24461.256,E2 -24461.256} C_VEL
LIN {X 0,Y 143.309,Z 340.353,A -85,B 0,C 180,E1 -24462.522,E2 -24462.522} C_VEL
LIN {X 0,Y 143.531,Z 340.053,A -85,B 0,C 180,E1 -24468.707,E2 -24468.707} C_VEL
LIN {X 0,Y 143.609,Z 340.046,A -85,B 0,C 180,E1 -24471.559,E2 -24471.559} C_VEL
LIN {X 0,Y 144.171,Z 339.967,A -85,B 0,C 180,E1 -24480.002,E2 -24480.002} C_VEL
LIN {X 0,Y 143.61,Z 340.04,A -85,B 0,C 180,E1 -24488.444,E2 -24488.444} C_VEL
LIN {X 0,Y 143.502,Z 340.063,A -85,B 0,C 180,E1 -24491.629,E2 -24491.629} C_VEL
LIN {X 0,Y 143.332,Z 340.389,A -85,B 0,C 180,E1 -24497.295,E2 -24497.295} C_VEL
LIN {X 0,Y 143.652,Z 341.626,A -85,B 0,C 180,E1 -24498.636,E2 -24498.636} C_VEL
LIN {X 0,Y 145.301,Z 344.224,A -85,B 0,C 180,E1 -24500.855,E2 -24500.855} C_VEL
LIN {X 0,Y 148.129,Z 346.357,A -85,B 0,C 180,E1 -24503.785,E2 -24503.785} C_VEL
LIN {X 0,Y 149.812,Z 349.232,A -85,B 0,C 180,E1 -24505.507,E2 -24505.507} C_VEL
LIN {X 0,Y 152.539,Z 351.758,A -85,B 0,C 180,E1 -24507.809,E2 -24507.809} C_VEL
LIN {X 0,Y 154.929,Z 355.248,A -85,B 0,C 180,E1 -24509.747,E2 -24509.747} C_VEL
LIN {X 0,Y 156.502,Z 356.974,A -85,B 0,C 180,E1 -24510.883,E2 -24510.883} C_VEL
LIN {X 0,Y 159.261,Z 360.683,A -85,B 0,C 180,E1 -24512.795,E2 -24512.795} C_VEL
LIN {X 0,Y 162.588,Z 365.615,A -85,B 0,C 180,E1 -24514.932,E2 -24514.932} C_VEL
LIN {X 0,Y 167.367,Z 374.225,A -85,B 0,C 180,E1 -24517.787,E2 -24517.787} C_VEL
LIN {X 0,Y 173.583,Z 387.164,A -85,B 0,C 180,E1 -24521.143,E2 -24521.143} C_VEL
LIN {X 0,Y 178.66,Z 399.849,A -85,B 0,C 180,E1 -24523.687,E2 -24523.687} C_VEL
LIN {X 0,Y 179.894,Z 403.845,A -85,B 0,C 180,E1 -24524.318,E2 -24524.318} C_VEL
LIN {X 0,Y 180.204,Z 408.171,A -85,B 0,C 180,E1 -24524.658,E2 -24524.658} C_VEL
LIN {X 0,Y 177.793,Z 443.25,A -85,B 0,C 180,E1 -24525.919,E2 -24525.919} C_VEL
LIN {X 0,Y 176.378,Z 454.418,A -85,B 0,C 180,E1 -24526.567,E2 -24526.567} C_VEL
LIN {X 0,Y 173.958,Z 467.037,A -85,B 0,C 180,E1 -24527.61,E2 -24527.61} C_VEL
LIN {X 0,Y 170.538,Z 479.743,A -85,B 0,C 180,E1 -24529.141,E2 -24529.141} C_VEL
LIN {X 0,Y 167.551,Z 489.013,A -85,B 0,C 180,E1 -24530.624,E2 -24530.624} C_VEL
LIN {X 0,Y 164.228,Z 497.952,A -85,B 0,C 180,E1 -24532.425,E2 -24532.425} C_VEL
LIN {X 0,Y 160.664,Z 506.475,A -85,B 0,C 180,E1 -24534.578,E2 -24534.578} C_VEL
LIN {X 0,Y 157.359,Z 513.69,A -85,B 0,C 180,E1 -24536.832,E2 -24536.832} C_VEL
LIN {X 0,Y 154.36,Z 519.889,A -85,B 0,C 180,E1 -24539.19,E2 -24539.19} C_VEL
LIN {X 0,Y 151.057,Z 526.427,A -85,B 0,C 180,E1 -24542.274,E2 -24542.274} C_VEL
LIN {X 0,Y 148.754,Z 530.931,A -85,B 0,C 180,E1 -24544.837,E2 -24544.837} C_VEL
LIN {X 0,Y 145.696,Z 536.422,A -85,B 0,C 180,E1 -24548.791,E2 -24548.791} C_VEL
LIN {X 0,Y 143.3,Z 540.748,A -85,B 0,C 180,E1 -24552.887,E2 -24552.887} C_VEL
LIN {X 0,Y 142.221,Z 543.121,A -85,B 0,C 180,E1 -24555.696,E2 -24555.696} C_VEL
LIN {X 0,Y 141.401,Z 544.925,A -85,B 0,C 180,E1 -24558.533,E2 -24558.533} C_VEL
LIN {X 0,Y 140.617,Z 547.386,A -85,B 0,C 180,E1 -24564.263,E2 -24564.263} C_VEL
LIN {X 0,Y 140.572,Z 548.139,A -85,B 0,C 180,E1 -24569.356,E2 -24569.356} C_VEL
LIN {X 0,Y 140.489,Z 547.98,A -85,B 0,C 180,E1 -24572.867,E2 -24572.867} C_VEL
LIN {X 0,Y 140.548,Z 547.384,A -85,B 0,C 180,E1 -24575.74,E2 -24575.74} C_VEL
LIN {X 0,Y 141.4,Z 544.925,A -85,B 0,C 180,E1 -24581.467,E2 -24581.467} C_VEL
LIN {X 0,Y 142.728,Z 541.967,A -85,B 0,C 180,E1 -24585.713,E2 -24585.713} C_VEL
LIN {X 0,Y 144.811,Z 537.975,A -85,B 0,C 180,E1 -24589.86,E2 -24589.86} C_VEL
LIN {X 0,Y 147.622,Z 532.845,A -85,B 0,C 180,E1 -24593.87,E2 -24593.87} C_VEL
LIN {X 0,Y 150.539,Z 527.586,A -85,B 0,C 180,E1 -24597.076,E2 -24597.076} C_VEL
LIN {X 0,Y 153.65,Z 521.265,A -85,B 0,C 180,E1 -24600.207,E2 -24600.207} C_VEL
LIN {X 0,Y 156.593,Z 515.316,A -85,B 0,C 180,E1 -24602.585,E2 -24602.585} C_VEL
LIN {X 0,Y 159.823,Z 508.394,A -85,B 0,C 180,E1 -24604.865,E2 -24604.865} C_VEL
LIN {X 0,Y 163.327,Z 500.22,A -85,B 0,C 180,E1 -24607.043,E2 -24607.043} C_VEL
LIN {X 0,Y 166.59,Z 491.715,A -85,B 0,C 180,E1 -24608.867,E2 -24608.867} C_VEL
LIN {X 0,Y 169.634,Z 482.507,A -85,B 0,C 180,E1 -24610.459,E2 -24610.459} C_VEL
LIN {X 0,Y 170.826,Z 477.345,A -85,B 0,C 180,E1 -24611.336,E2 -24611.336} C_VEL
LIN {X 0,Y 171.02,Z 468.718,A -85,B 0,C 180,E1 -24612.975,E2 -24612.975} C_VEL
LIN {X 0,Y 170.915,Z 459.855,A -85,B 0,C 180,E1 -24614.462,E2 -24614.462} C_VEL
LIN {X 0,Y 171.301,Z 454.232,A -85,B 0,C 180,E1 -24615.062,E2 -24615.062} C_VEL
LIN {X 0,Y 172.72,Z 443.746,A -85,B 0,C 180,E1 -24615.67,E2 -24615.67} C_VEL
LIN {X 0,Y 174.955,Z 412.719,A -85,B 0,C 180,E1 -24616.83,E2 -24616.83} C_VEL
LIN {X 0,Y 175.165,Z 407.044,A -85,B 0,C 180,E1 -24617.09,E2 -24617.09} C_VEL
LIN {X 0,Y 173.907,Z 402.814,A -85,B 0,C 180,E1 -24617.788,E2 -24617.788} C_VEL
LIN {X 0,Y 169.057,Z 390.302,A -85,B 0,C 180,E1 -24620.428,E2 -24620.428} C_VEL
LIN {X 0,Y 163.277,Z 378.139,A -85,B 0,C 180,E1 -24623.806,E2 -24623.806} C_VEL
LIN {X 0,Y 159.03,Z 370.259,A -85,B 0,C 180,E1 -24626.561,E2 -24626.561} C_VEL
LIN {X 0,Y 155.995,Z 365.936,A -85,B 0,C 180,E1 -24628.646,E2 -24628.646} C_VEL
LIN {X 0,Y 153.181,Z 362.073,A -85,B 0,C 180,E1 -24630.764,E2 -24630.764} C_VEL
LIN {X 0,Y 150.361,Z 358.194,A -85,B 0,C 180,E1 -24633.125,E2 -24633.125} C_VEL
LIN {X 0,Y 147.031,Z 354.536,A -85,B 0,C 180,E1 -24636.213,E2 -24636.213} C_VEL
LIN {X 0,Y 146.021,Z 352.666,A -85,B 0,C 180,E1 -24637.352,E2 -24637.352} C_VEL
LIN {X 0,Y 143.256,Z 350.351,A -85,B 0,C 180,E1 -24640.474,E2 -24640.474} C_VEL
LIN {X 0,Y 141.536,Z 347.232,A -85,B 0,C 180,E1 -24643.037,E2 -24643.037} C_VEL
LIN {X 0,Y 138.37,Z 344.922,A -85,B 0,C 180,E1 -24648.549,E2 -24648.549} C_VEL
LIN {X 0,Y 136.719,Z 341.69,A -85,B 0,C 180,E1 -24654.837,E2 -24654.837} C_VEL
LIN {X 0,Y 137.128,Z 340.975,A -85,B 0,C 180,E1 -24659.998,E2 -24659.998} C_VEL
LIN {X 0,Y 136.7,Z 341.612,A -85,B 0,C 180,E1 -24665.16,E2 -24665.16} C_VEL
LIN {X 0,Y 137.44,Z 343.666,A -85,B 0,C 180,E1 -24669.379,E2 -24669.379} C_VEL
LIN {X 0,Y 139.939,Z 346.365,A -85,B 0,C 180,E1 -24674.913,E2 -24674.913} C_VEL
LIN {X 0,Y 141.64,Z 347.359,A -85,B 0,C 180,E1 -24677.505,E2 -24677.505} C_VEL
LIN {X 0,Y 143.247,Z 350.329,A -85,B 0,C 180,E1 -24679.898,E2 -24679.898} C_VEL
LIN {X 0,Y 145.387,Z 352.307,A -85,B 0,C 180,E1 -24682.386,E2 -24682.386} C_VEL
LIN {X 0,Y 146.23,Z 352.98,A -85,B 0,C 180,E1 -24683.264,E2 -24683.264} C_VEL
LIN {X 0,Y 148.37,Z 356.271,A -85,B 0,C 180,E1 -24685.501,E2 -24685.501} C_VEL
LIN {X 0,Y 150.389,Z 358.229,A -85,B 0,C 180,E1 -24687.283,E2 -24687.283} C_VEL
LIN {X 0,Y 152.963,Z 361.853,A -85,B 0,C 180,E1 -24689.455,E2 -24689.455} C_VEL
LIN {X 0,Y 154.37,Z 363.661,A -85,B 0,C 180,E1 -24690.537,E2 -24690.537} C_VEL
LIN {X 0,Y 157.872,Z 368.542,A -85,B 0,C 180,E1 -24693.046,E2 -24693.046} C_VEL
LIN {X 0,Y 162.422,Z 375.14,A -85,B 0,C 180,E1 -24695.945,E2 -24695.945} C_VEL
LIN {X 0,Y 168.769,Z 385.702,A -85,B 0,C 180,E1 -24699.538,E2 -24699.538} C_VEL
LIN {X 0,Y 174.554,Z 396.667,A -85,B 0,C 180,E1 -24702.461,E2 -24702.461} C_VEL
LIN {X 0,Y 180.342,Z 409.898,A -85,B 0,C 180,E1 -24705.182,E2 -24705.182} C_VEL
LIN {X 0,Y 187.382,Z 426.74,A -85,B 0,C 180,E1 -24708.154,E2 -24708.154} C_VEL
LIN {X 0,Y 194.669,Z 440.906,A -85,B 0,C 180,E1 -24710.912,E2 -24710.912} C_VEL
LIN {X 0,Y 201.422,Z 452.735,A -85,B 0,C 180,E1 -24713.619,E2 -24713.619} C_VEL
LIN {X 0,Y 208.629,Z 463.399,A -85,B 0,C 180,E1 -24716.428,E2 -24716.428} C_VEL
LIN {X 0,Y 216.494,Z 473.398,A -85,B 0,C 180,E1 -24719.344,E2 -24719.344} C_VEL
LIN {X 0,Y 225.764,Z 483.338,A -85,B 0,C 180,E1 -24722.519,E2 -24722.519} C_VEL
LIN {X 0,Y 235.536,Z 491.846,A -85,B 0,C 180,E1 -24725.51,E2 -24725.51} C_VEL
LIN {X 0,Y 248.447,Z 500.92,A -85,B 0,C 180,E1 -24728.984,E2 -24728.984} C_VEL
LIN {X 0,Y 262.84,Z 509.475,A -85,B 0,C 180,E1 -24732.495,E2 -24732.495} C_VEL
LIN {X 0,Y 273.631,Z 515.61,A -85,B 0,C 180,E1 -24735.118,E2 -24735.118} C_VEL
LIN {X 0,Y 281.164,Z 520.123,A -85,B 0,C 180,E1 -24737.118,E2 -24737.118} C_VEL
LIN {X 0,Y 289.301,Z 525.022,A -85,B 0,C 180,E1 -24739.508,E2 -24739.508} C_VEL
LIN {X 0,Y 292.153,Z 526.802,A -85,B 0,C 180,E1 -24740.496,E2 -24740.496} C_VEL
LIN {X 0,Y 295.201,Z 528.9,A -85,B 0,C 180,E1 -24741.788,E2 -24741.788} C_VEL
LIN {X 0,Y 298.242,Z 530.849,A -85,B 0,C 180,E1 -24743.234,E2 -24743.234} C_VEL
LIN {X 0,Y 300.699,Z 532.211,A -85,B 0,C 180,E1 -24744.636,E2 -24744.636} C_VEL
LIN {X 0,Y 302.913,Z 533.262,A -85,B 0,C 180,E1 -24746.067,E2 -24746.067} C_VEL
LIN {X 0,Y 304.424,Z 533.934,A -85,B 0,C 180,E1 -24747.354,E2 -24747.354} C_VEL
LIN {X 0,Y 305.376,Z 534.327,A -85,B 0,C 180,E1 -24748.681,E2 -24748.681} C_VEL
LIN {X 0,Y 305.851,Z 534.413,A -85,B 0,C 180,E1 -24750,E2 -24750} C_VEL
LIN {X 0,Y 305.42,Z 534.32,A -85,B 0,C 180,E1 -24751.319,E2 -24751.319} C_VEL
LIN {X 0,Y 304.449,Z 533.938,A -85,B 0,C 180,E1 -24752.646,E2 -24752.646} C_VEL
LIN {X 0,Y 302.814,Z 533.248,A -85,B 0,C 180,E1 -24753.992,E2 -24753.992} C_VEL
LIN {X 0,Y 300.739,Z 532.234,A -85,B 0,C 180,E1 -24755.363,E2 -24755.363} C_VEL
LIN {X 0,Y 297.472,Z 530.401,A -85,B 0,C 180,E1 -24757.13,E2 -24757.13} C_VEL
LIN {X 0,Y 293.744,Z 527.893,A -85,B 0,C 180,E1 -24758.851,E2 -24758.851} C_VEL
LIN {X 0,Y 291.62,Z 526.435,A -85,B 0,C 180,E1 -24759.712,E2 -24759.712} C_VEL
LIN {X 0,Y 286.682,Z 523.393,A -85,B 0,C 180,E1 -24761.31,E2 -24761.31} C_VEL
LIN {X 0,Y 278.185,Z 518.293,A -85,B 0,C 180,E1 -24763.702,E2 -24763.702} C_VEL
LIN {X 0,Y 270.151,Z 513.669,A -85,B 0,C 180,E1 -24765.732,E2 -24765.732} C_VEL
LIN {X 0,Y 259.185,Z 507.423,A -85,B 0,C 180,E1 -24768.371,E2 -24768.371} C_VEL
LIN {X 0,Y 246.73,Z 499.783,A -85,B 0,C 180,E1 -24771.458,E2 -24771.458} C_VEL
LIN {X 0,Y 234.431,Z 490.931,A -85,B 0,C 180,E1 -24774.815,E2 -24774.815} C_VEL
LIN {X 0,Y 223.408,Z 480.975,A -85,B 0,C 180,E1 -24778.26,E2 -24778.26} C_VEL
LIN {X 0,Y 214.254,Z 470.714,A -85,B 0,C 180,E1 -24781.479,E2 -24781.479} C_VEL
LIN {X 0,Y 206.191,Z 459.871,A -85,B 0,C 180,E1 -24784.539,E2 -24784.539} C_VEL
LIN {X 0,Y 199.116,Z 448.805,A -85,B 0,C 180,E1 -24787.322,E2 -24787.322} C_VEL
LIN {X 0,Y 192.468,Z 436.802,A -85,B 0,C 180,E1 -24789.933,E2 -24789.933} C_VEL
LIN {X 0,Y 185.929,Z 423.591,A -85,B 0,C 180,E1 -24792.413,E2 -24792.413} C_VEL
LIN {X 0,Y 177.526,Z 403.271,A -85,B 0,C 180,E1 -24796.114,E2 -24796.114} C_VEL
LIN {X 0,Y 172.671,Z 392.926,A -85,B 0,C 180,E1 -24798.461,E2 -24798.461} C_VEL
LIN {X 0,Y 167.444,Z 383.424,A -85,B 0,C 180,E1 -24801.172,E2 -24801.172} C_VEL
LIN {X 0,Y 161.9,Z 374.35,A -85,B 0,C 180,E1 -24804.371,E2 -24804.371} C_VEL
LIN {X 0,Y 156.74,Z 366.813,A -85,B 0,C 180,E1 -24807.747,E2 -24807.747} C_VEL
LIN {X 0,Y 153.303,Z 362.203,A -85,B 0,C 180,E1 -24810.287,E2 -24810.287} C_VEL
LIN {X 0,Y 150.557,Z 358.553,A -85,B 0,C 180,E1 -24812.558,E2 -24812.558} C_VEL
LIN {X 0,Y 149.98,Z 357.73,A -85,B 0,C 180,E1 -24813.076,E2 -24813.076} C_VEL
LIN {X 0,Y 147.369,Z 355.022,A -85,B 0,C 180,E1 -24815.479,E2 -24815.479} C_VEL
LIN {X 0,Y 146.01,Z 352.653,A -85,B 0,C 180,E1 -24816.98,E2 -24816.98} C_VEL
LIN {X 0,Y 143.525,Z 350.682,A -85,B 0,C 180,E1 -24819.745,E2 -24819.745} C_VEL
LIN {X 0,Y 141.797,Z 347.709,A -85,B 0,C 180,E1 -24822.236,E2 -24822.236} C_VEL
LIN {X 0,Y 140.822,Z 346.801,A -85,B 0,C 180,E1 -24823.698,E2 -24823.698} C_VEL
LIN {X 0,Y 138.204,Z 344.776,A -85,B 0,C 180,E1 -24828.54,E2 -24828.54} C_VEL
LIN {X 0,Y 136.71,Z 341.85,A -85,B 0,C 180,E1 -24834.1,E2 -24834.1} C_VEL
LIN {X 0,Y 136.786,Z 341.203,A -85,B 0,C 180,E1 -24837.057,E2 -24837.057} C_VEL
LIN {X 0,Y 137.128,Z 340.973,A -85,B 0,C 180,E1 -24840.002,E2 -24840.002} C_VEL
LIN {X 0,Y 136.719,Z 341.705,A -85,B 0,C 180,E1 -24845.163,E2 -24845.163} C_VEL
LIN {X 0,Y 139.948,Z 346.364,A -85,B 0,C 180,E1 -24854.544,E2 -24854.544} C_VEL
LIN {X 0,Y 141.647,Z 347.392,A -85,B 0,C 180,E1 -24857.135,E2 -24857.135} C_VEL
LIN {X 0,Y 143.387,Z 350.509,A -85,B 0,C 180,E1 -24859.694,E2 -24859.694} C_VEL
LIN {X 0,Y 146.021,Z 352.664,A -85,B 0,C 180,E1 -24862.648,E2 -24862.648} C_VEL
LIN {X 0,Y 148.142,Z 356.025,A -85,B 0,C 180,E1 -24864.902,E2 -24864.902} C_VEL
LIN {X 0,Y 150.481,Z 358.406,A -85,B 0,C 180,E1 -24866.986,E2 -24866.986} C_VEL
LIN {X 0,Y 153.183,Z 362.063,A -85,B 0,C 180,E1 -24869.236,E2 -24869.236} C_VEL
LIN {X 0,Y 157.609,Z 368.168,A -85,B 0,C 180,E1 -24872.482,E2 -24872.482} C_VEL
LIN {X 0,Y 159.76,Z 371.63,A -85,B 0,C 180,E1 -24873.938,E2 -24873.938} C_VEL
LIN {X 0,Y 163.934,Z 379.441,A -85,B 0,C 180,E1 -24876.598,E2 -24876.598} C_VEL
LIN {X 0,Y 170.154,Z 392.883,A -85,B 0,C 180,E1 -24880.18,E2 -24880.18} C_VEL
LIN {X 0,Y 174.733,Z 405.186,A -85,B 0,C 180,E1 -24882.648,E2 -24882.648} C_VEL
LIN {X 0,Y 175.233,Z 407.957,A -85,B 0,C 180,E1 -24882.987,E2 -24882.987} C_VEL
LIN {X 0,Y 172.673,Z 443.975,A -85,B 0,C 180,E1 -24884.325,E2 -24884.325} C_VEL
LIN {X 0,Y 170.967,Z 456.447,A -85,B 0,C 180,E1 -24885.089,E2 -24885.089} C_VEL
LIN {X 0,Y 167.936,Z 470.039,A -85,B 0,C 180,E1 -24886.33,E2 -24886.33} C_VEL
LIN {X 0,Y 165.244,Z 479.549,A -85,B 0,C 180,E1 -24887.533,E2 -24887.533} C_VEL
LIN {X 0,Y 162.132,Z 488.82,A -85,B 0,C 180,E1 -24889.034,E2 -24889.034} C_VEL
LIN {X 0,Y 158.662,Z 497.758,A -85,B 0,C 180,E1 -24890.862,E2 -24890.862} C_VEL
LIN {X 0,Y 154.932,Z 506.281,A -85,B 0,C 180,E1 -24893.056,E2 -24893.056} C_VEL
LIN {X 0,Y 151.438,Z 513.495,A -85,B 0,C 180,E1 -24895.355,E2 -24895.355} C_VEL
LIN {X 0,Y 148.279,Z 519.695,A -85,B 0,C 180,E1 -24897.778,E2 -24897.778} C_VEL
LIN {X 0,Y 144.735,Z 526.231,A -85,B 0,C 180,E1 -24900.951,E2 -24900.951} C_VEL
LIN {X 0,Y 142.358,Z 530.737,A -85,B 0,C 180,E1 -24903.621,E2 -24903.621} C_VEL
LIN {X 0,Y 139.075,Z 536.227,A -85,B 0,C 180,E1 -24907.729,E2 -24907.729} C_VEL
LIN {X 0,Y 136.495,Z 540.553,A -85,B 0,C 180,E1 -24912.005,E2 -24912.005} C_VEL
LIN {X 0,Y 135.328,Z 542.926,A -85,B 0,C 180,E1 -24914.95,E2 -24914.95} C_VEL
LIN {X 0,Y 134.436,Z 544.731,A -85,B 0,C 180,E1 -24917.93,E2 -24917.93} C_VEL
LIN {X 0,Y 133.542,Z 547.191,A -85,B 0,C 180,E1 -24923.958,E2 -24923.958} C_VEL
LIN {X 0,Y 133.414,Z 547.786,A -85,B 0,C 180,E1 -24926.98,E2 -24926.98} C_VEL
LIN {X 0,Y 133.536,Z 547.947,A -85,B 0,C 180,E1 -24930,E2 -24930} C_VEL
LIN {X 0,Y 133.4,Z 547.786,A -85,B 0,C 180,E1 -24933.02,E2 -24933.02} C_VEL
LIN {X 0,Y 133.466,Z 547.189,A -85,B 0,C 180,E1 -24936.045,E2 -24936.045} C_VEL
LIN {X 0,Y 134.435,Z 544.731,A -85,B 0,C 180,E1 -24942.07,E2 -24942.07} C_VEL
LIN {X 0,Y 135.869,Z 541.772,A -85,B 0,C 180,E1 -24946.528,E2 -24946.528} C_VEL
LIN {X 0,Y 138.124,Z 537.781,A -85,B 0,C 180,E1 -24950.865,E2 -24950.865} C_VEL
LIN {X 0,Y 141.137,Z 532.65,A -85,B 0,C 180,E1 -24955.04,E2 -24955.04} C_VEL
LIN {X 0,Y 144.212,Z 527.402,A -85,B 0,C 180,E1 -24958.361,E2 -24958.361} C_VEL
LIN {X 0,Y 147.53,Z 521.07,A -85,B 0,C 180,E1 -24961.601,E2 -24961.601} C_VEL
LIN {X 0,Y 150.63,Z 515.122,A -85,B 0,C 180,E1 -24964.047,E2 -24964.047} C_VEL
LIN {X 0,Y 154.045,Z 508.2,A -85,B 0,C 180,E1 -24966.376,E2 -24966.376} C_VEL
LIN {X 0,Y 157.705,Z 500.026,A -85,B 0,C 180,E1 -24968.6,E2 -24968.6} C_VEL
LIN {X 0,Y 161.119,Z 491.521,A -85,B 0,C 180,E1 -24970.453,E2 -24970.453} C_VEL
LIN {X 0,Y 164.184,Z 482.685,A -85,B 0,C 180,E1 -24972.008,E2 -24972.008} C_VEL
LIN {X 0,Y 167.091,Z 473.058,A -85,B 0,C 180,E1 -24973.322,E2 -24973.322} C_VEL
LIN {X 0,Y 169.306,Z 464.27,A -85,B 0,C 180,E1 -24974.257,E2 -24974.257} C_VEL
LIN {X 0,Y 171.301,Z 454.232,A -85,B 0,C 180,E1 -24975.062,E2 -24975.062} C_VEL
LIN {X 0,Y 171.708,Z 448.543,A -85,B 0,C 180,E1 -24975.601,E2 -24975.601} C_VEL
LIN {X 0,Y 169.41,Z 429.956,A -85,B 0,C 180,E1 -24977.792,E2 -24977.792} C_VEL
LIN {X 0,Y 169.367,Z 424.151,A -85,B 0,C 180,E1 -24978.157,E2 -24978.157} C_VEL
LIN {X 0,Y 170.336,Z 408.821,A -85,B 0,C 180,E1 -24978.744,E2 -24978.744} C_VEL
LIN {X 0,Y 165.704,Z 396.084,A -85,B 0,C 180,E1 -24981.448,E2 -24981.448} C_VEL
LIN {X 0,Y 159.94,Z 383.28,A -85,B 0,C 180,E1 -24985.066,E2 -24985.066} C_VEL
LIN {X 0,Y 155.856,Z 375.541,A -85,B 0,C 180,E1 -24987.908,E2 -24987.908} C_VEL
LIN {X 0,Y 152.823,Z 371.115,A -85,B 0,C 180,E1 -24990.16,E2 -24990.16} C_VEL
LIN {X 0,Y 150.712,Z 368.078,A -85,B 0,C 180,E1 -24991.876,E2 -24991.876} C_VEL
LIN {X 0,Y 147.64,Z 363.916,A -85,B 0,C 180,E1 -24994.631,E2 -24994.631} C_VEL
LIN {X 0,Y 144.856,Z 360.502,A -85,B 0,C 180,E1 -24997.466,E2 -24997.466} C_VEL
LIN {X 0,Y 143.99,Z 359.167,A -85,B 0,C 180,E1 -24998.479,E2 -24998.479} C_VEL
LIN {X 0,Y 141.358,Z 356.49,A -85,B 0,C 180,E1 -25001.754,E2 -25001.754} C_VEL
LIN {X 0,Y 139.992,Z 353.912,A -85,B 0,C 180,E1 -25003.97,E2 -25003.97} C_VEL
LIN {X 0,Y 137.266,Z 351.852,A -85,B 0,C 180,E1 -25009.035,E2 -25009.035} C_VEL
LIN {X 0,Y 135.523,Z 348.555,A -85,B 0,C 180,E1 -25015.537,E2 -25015.537} C_VEL
LIN {X 0,Y 135.17,Z 347.795,A -85,B 0,C 180,E1 -25019.998,E2 -25019.998} C_VEL
LIN {X 0,Y 135.581,Z 348.666,A -85,B 0,C 180,E1 -25025.203,E2 -25025.203} C_VEL
LIN {X 0,Y 138.587,Z 353.166,A -85,B 0,C 180,E1 -25034.124,E2 -25034.124} C_VEL
LIN {X 0,Y 140.197,Z 354.206,A -85,B 0,C 180,E1 -25036.751,E2 -25036.751} C_VEL
LIN {X 0,Y 142.12,Z 357.534,A -85,B 0,C 180,E1 -25039.686,E2 -25039.686} C_VEL
LIN {X 0,Y 144.441,Z 359.661,A -85,B 0,C 180,E1 -25042.414,E2 -25042.414} C_VEL
LIN {X 0,Y 146.785,Z 363.119,A -85,B 0,C 180,E1 -25044.955,E2 -25044.955} C_VEL
LIN {X 0,Y 148.325,Z 364.716,A -85,B 0,C 180,E1 -25046.387,E2 -25046.387} C_VEL
LIN {X 0,Y 151.034,Z 368.45,A -85,B 0,C 180,E1 -25048.77,E2 -25048.77} C_VEL
LIN {X 0,Y 155.351,Z 374.724,A -85,B 0,C 180,E1 -25052.11,E2 -25052.11} C_VEL
LIN {X 0,Y 159.32,Z 380.671,A -85,B 0,C 180,E1 -25054.798,E2 -25054.798} C_VEL
LIN {X 0,Y 165.423,Z 391.153,A -85,B 0,C 180,E1 -25058.477,E2 -25058.477} C_VEL
LIN {X 0,Y 171.227,Z 402.705,A -85,B 0,C 180,E1 -25061.598,E2 -25061.598} C_VEL
LIN {X 0,Y 176.456,Z 415.347,A -85,B 0,C 180,E1 -25064.218,E2 -25064.218} C_VEL
LIN {X 0,Y 182.882,Z 431.046,A -85,B 0,C 180,E1 -25067.099,E2 -25067.099} C_VEL
LIN {X 0,Y 188.87,Z 443.571,A -85,B 0,C 180,E1 -25069.712,E2 -25069.712} C_VEL
LIN {X 0,Y 193.911,Z 452.978,A -85,B 0,C 180,E1 -25071.966,E2 -25071.966} C_VEL
LIN {X 0,Y 199.108,Z 461.67,A -85,B 0,C 180,E1 -25074.274,E2 -25074.274} C_VEL
LIN {X 0,Y 206.157,Z 471.756,A -85,B 0,C 180,E1 -25077.274,E2 -25077.274} C_VEL
LIN {X 0,Y 213.186,Z 480.346,A -85,B 0,C 180,E1 -25080.062,E2 -25080.062} C_VEL
LIN {X 0,Y 222.557,Z 489.902,A -85,B 0,C 180,E1 -25083.453,E2 -25083.453} C_VEL
LIN {X 0,Y 234.066,Z 499.003,A -85,B 0,C 180,E1 -25087.025,E2 -25087.025} C_VEL
LIN {X 0,Y 246.27,Z 506.801,A -85,B 0,C 180,E1 -25090.344,E2 -25090.344} C_VEL
LIN {X 0,Y 259.12,Z 513.912,A -85,B 0,C 180,E1 -25093.557,E2 -25093.557} C_VEL
LIN {X 0,Y 268.199,Z 518.703,A -85,B 0,C 180,E1 -25095.824,E2 -25095.824} C_VEL
LIN {X 0,Y 273.741,Z 521.724,A -85,B 0,C 180,E1 -25097.315,E2 -25097.315} C_VEL
LIN {X 0,Y 279.292,Z 524.828,A -85,B 0,C 180,E1 -25098.922,E2 -25098.922} C_VEL
LIN {X 0,Y 284.874,Z 527.915,A -85,B 0,C 180,E1 -25100.682,E2 -25100.682} C_VEL
LIN {X 0,Y 288.81,Z 530.441,A -85,B 0,C 180,E1 -25102.309,E2 -25102.309} C_VEL
LIN {X 0,Y 290.366,Z 531.474,A -85,B 0,C 180,E1 -25103.049,E2 -25103.049} C_VEL
LIN {X 0,Y 293.097,Z 533.068,A -85,B 0,C 180,E1 -25104.496,E2 -25104.496} C_VEL
LIN {X 0,Y 295.828,Z 534.461,A -85,B 0,C 180,E1 -25106.18,E2 -25106.18} C_VEL
LIN {X 0,Y 297.186,Z 535.085,A -85,B 0,C 180,E1 -25107.289,E2 -25107.289} C_VEL
LIN {X 0,Y 298.3,Z 535.503,A -85,B 0,C 180,E1 -25108.65,E2 -25108.65} C_VEL
LIN {X 0,Y 298.86,Z 535.605,A -85,B 0,C 180,E1 -25110,E2 -25110} C_VEL
LIN {X 0,Y 298.336,Z 535.504,A -85,B 0,C 180,E1 -25111.35,E2 -25111.35} C_VEL
LIN {X 0,Y 297.205,Z 535.098,A -85,B 0,C 180,E1 -25112.711,E2 -25112.711} C_VEL
LIN {X 0,Y 295.399,Z 534.296,A -85,B 0,C 180,E1 -25114.093,E2 -25114.093} C_VEL
LIN {X 0,Y 293.125,Z 533.073,A -85,B 0,C 180,E1 -25115.503,E2 -25115.503} C_VEL
LIN {X 0,Y 290.289,Z 531.455,A -85,B 0,C 180,E1 -25116.97,E2 -25116.97} C_VEL
LIN {X 0,Y 287.069,Z 529.326,A -85,B 0,C 180,E1 -25118.447,E2 -25118.447} C_VEL
LIN {X 0,Y 282.813,Z 526.706,A -85,B 0,C 180,E1 -25120.017,E2 -25120.017} C_VEL
LIN {X 0,Y 277.195,Z 523.659,A -85,B 0,C 180,E1 -25121.702,E2 -25121.702} C_VEL
LIN {X 0,Y 268.197,Z 518.707,A -85,B 0,C 180,E1 -25124.175,E2 -25124.175} C_VEL
LIN {X 0,Y 257.124,Z 512.852,A -85,B 0,C 180,E1 -25126.934,E2 -25126.934} C_VEL
LIN {X 0,Y 244.152,Z 505.534,A -85,B 0,C 180,E1 -25130.207,E2 -25130.207} C_VEL
LIN {X 0,Y 232.109,Z 497.595,A -85,B 0,C 180,E1 -25133.545,E2 -25133.545} C_VEL
LIN {X 0,Y 221.024,Z 488.444,A -85,B 0,C 180,E1 -25137.088,E2 -25137.088} C_VEL
LIN {X 0,Y 211.912,Z 478.916,A -85,B 0,C 180,E1 -25140.429,E2 -25140.429} C_VEL
LIN {X 0,Y 203.269,Z 467.907,A -85,B 0,C 180,E1 -25143.924,E2 -25143.924} C_VEL
LIN {X 0,Y 197.042,Z 458.406,A -85,B 0,C 180,E1 -25146.631,E2 -25146.631} C_VEL
LIN {X 0,Y 190.528,Z 446.796,A -85,B 0,C 180,E1 -25149.543,E2 -25149.543} C_VEL
LIN {X 0,Y 185.005,Z 435.615,A -85,B 0,C 180,E1 -25152.002,E2 -25152.002} C_VEL
LIN {X 0,Y 177.885,Z 419.216,A -85,B 0,C 180,E1 -25155.09,E2 -25155.09} C_VEL
LIN {X 0,Y 173.277,Z 407.527,A -85,B 0,C 180,E1 -25157.348,E2 -25157.348} C_VEL
LIN {X 0,Y 168.749,Z 397.549,A -85,B 0,C 180,E1 -25159.698,E2 -25159.698} C_VEL
LIN {X 0,Y 163.855,Z 388.366,A -85,B 0,C 180,E1 -25162.419,E2 -25162.419} C_VEL
LIN {X 0,Y 158.781,Z 379.852,A -85,B 0,C 180,E1 -25165.549,E2 -25165.549} C_VEL
LIN {X 0,Y 154.213,Z 372.898,A -85,B 0,C 180,E1 -25168.737,E2 -25168.737} C_VEL
LIN {X 0,Y 150.752,Z 368.15,A -85,B 0,C 180,E1 -25171.457,E2 -25171.457} C_VEL
LIN {X 0,Y 147.657,Z 363.926,A -85,B 0,C 180,E1 -25174.232,E2 -25174.232} C_VEL
LIN {X 0,Y 145.085,Z 360.844,A -85,B 0,C 180,E1 -25176.824,E2 -25176.824} C_VEL
LIN {X 0,Y 144.11,Z 359.244,A -85,B 0,C 180,E1 -25177.965,E2 -25177.965} C_VEL
LIN {X 0,Y 141.62,Z 356.872,A -85,B 0,C 180,E1 -25180.996,E2 -25180.996} C_VEL
LIN {X 0,Y 139.983,Z 353.919,A -85,B 0,C 180,E1 -25183.598,E2 -25183.598} C_VEL
LIN {X 0,Y 137.226,Z 351.857,A -85,B 0,C 180,E1 -25188.734,E2 -25188.734} C_VEL
LIN {X 0,Y 135.518,Z 348.573,A -85,B 0,C 180,E1 -25195.167,E2 -25195.167} C_VEL
LIN {X 0,Y 135.169,Z 347.803,A -85,B 0,C 180,E1 -25200.002,E2 -25200.002} C_VEL
LIN {X 0,Y 135.645,Z 348.82,A -85,B 0,C 180,E1 -25205.204,E2 -25205.204} C_VEL
LIN {X 0,Y 138.694,Z 353.229,A -85,B 0,C 180,E1 -25213.929,E2 -25213.929} C_VEL
LIN {X 0,Y 140.203,Z 354.225,A -85,B 0,C 180,E1 -25216.379,E2 -25216.379} C_VEL
LIN {X 0,Y 142.004,Z 357.353,A -85,B 0,C 180,E1 -25219.142,E2 -25219.142} C_VEL
LIN {X 0,Y 144.522,Z 359.821,A -85,B 0,C 180,E1 -25222.129,E2 -25222.129} C_VEL
LIN {X 0,Y 146.864,Z 363.174,A -85,B 0,C 180,E1 -25224.644,E2 -25224.644} C_VEL
LIN {X 0,Y 148.411,Z 364.869,A -85,B 0,C 180,E1 -25226.086,E2 -25226.086} C_VEL
LIN {X 0,Y 151.98,Z 369.883,A -85,B 0,C 180,E1 -25229.169,E2 -25229.169} C_VEL
LIN {X 0,Y 155.66,Z 375.171,A -85,B 0,C 180,E1 -25231.946,E2 -25231.946} C_VEL
LIN {X 0,Y 160.052,Z 383.427,A -85,B 0,C 180,E1 -25235.002,E2 -25235.002} C_VEL
LIN {X 0,Y 166.152,Z 397.164,A -85,B 0,C 180,E1 -25238.817,E2 -25238.817} C_VEL
LIN {X 0,Y 170.334,Z 408.869,A -85,B 0,C 180,E1 -25241.258,E2 -25241.258} C_VEL
LIN {X 0,Y 169.123,Z 427.293,A -85,B 0,C 180,E1 -25241.947,E2 -25241.947} C_VEL
LIN {X 0,Y 167.514,Z 446.667,A -85,B 0,C 180,E1 -25242.737,E2 -25242.737} C_VEL
LIN {X 0,Y 165.176,Z 460.215,A -85,B 0,C 180,E1 -25243.672,E2 -25243.672} C_VEL
LIN {X 0,Y 162.593,Z 470.852,A -85,B 0,C 180,E1 -25244.725,E2 -25244.725} C_VEL
LIN {X 0,Y 159.531,Z 480.986,A -85,B 0,C 180,E1 -25246.065,E2 -25246.065} C_VEL
LIN {X 0,Y 156.288,Z 489.976,A -85,B 0,C 180,E1 -25247.584,E2 -25247.584} C_VEL
LIN {X 0,Y 152.709,Z 498.698,A -85,B 0,C 180,E1 -25249.455,E2 -25249.455} C_VEL
LIN {X 0,Y 149.298,Z 506.087,A -85,B 0,C 180,E1 -25251.412,E2 -25251.412} C_VEL
LIN {X 0,Y 145.645,Z 513.301,A -85,B 0,C 180,E1 -25253.765,E2 -25253.765} C_VEL
LIN {X 0,Y 142.308,Z 519.5,A -85,B 0,C 180,E1 -25256.25,E2 -25256.25} C_VEL
LIN {X 0,Y 138.313,Z 526.43,A -85,B 0,C 180,E1 -25259.75,E2 -25259.75} C_VEL
LIN {X 0,Y 136.027,Z 530.543,A -85,B 0,C 180,E1 -25262.291,E2 -25262.291} C_VEL
LIN {X 0,Y 132.507,Z 536.032,A -85,B 0,C 180,E1 -25266.561,E2 -25266.561} C_VEL
LIN {X 0,Y 129.726,Z 540.358,A -85,B 0,C 180,E1 -25271.032,E2 -25271.032} C_VEL
LIN {X 0,Y 128.446,Z 542.731,A -85,B 0,C 180,E1 -25274.123,E2 -25274.123} C_VEL
LIN {X 0,Y 127.466,Z 544.536,A -85,B 0,C 180,E1 -25277.259,E2 -25277.259} C_VEL
LIN {X 0,Y 126.463,Z 546.997,A -85,B 0,C 180,E1 -25283.619,E2 -25283.619} C_VEL
LIN {X 0,Y 126.317,Z 547.592,A -85,B 0,C 180,E1 -25286.811,E2 -25286.811} C_VEL
LIN {X 0,Y 126.431,Z 547.753,A -85,B 0,C 180,E1 -25290,E2 -25290} C_VEL
LIN {X 0,Y 126.306,Z 547.592,A -85,B 0,C 180,E1 -25293.19,E2 -25293.19} C_VEL
LIN {X 0,Y 126.409,Z 546.995,A -85,B 0,C 180,E1 -25296.384,E2 -25296.384} C_VEL
LIN {X 0,Y 127.465,Z 544.536,A -85,B 0,C 180,E1 -25302.741,E2 -25302.741} C_VEL
LIN {X 0,Y 129.048,Z 541.578,A -85,B 0,C 180,E1 -25307.429,E2 -25307.429} C_VEL
LIN {X 0,Y 131.49,Z 537.586,A -85,B 0,C 180,E1 -25311.971,E2 -25311.971} C_VEL
LIN {X 0,Y 134.725,Z 532.456,A -85,B 0,C 180,E1 -25316.321,E2 -25316.321} C_VEL
LIN {X 0,Y 137.986,Z 527.137,A -85,B 0,C 180,E1 -25319.816,E2 -25319.816} C_VEL
LIN {X 0,Y 141.508,Z 520.876,A -85,B 0,C 180,E1 -25323.114,E2 -25323.114} C_VEL
LIN {X 0,Y 144.789,Z 514.927,A -85,B 0,C 180,E1 -25325.624,E2 -25325.624} C_VEL
LIN {X 0,Y 148.379,Z 508.005,A -85,B 0,C 180,E1 -25328.005,E2 -25328.005} C_VEL
LIN {X 0,Y 152.21,Z 499.832,A -85,B 0,C 180,E1 -25330.271,E2 -25330.271} C_VEL
LIN {X 0,Y 155.769,Z 491.327,A -85,B 0,C 180,E1 -25332.153,E2 -25332.153} C_VEL
LIN {X 0,Y 158.949,Z 482.616,A -85,B 0,C 180,E1 -25333.697,E2 -25333.697} C_VEL
LIN {X 0,Y 162.002,Z 472.864,A -85,B 0,C 180,E1 -25335.044,E2 -25335.044} C_VEL
LIN {X 0,Y 164.301,Z 464.076,A -85,B 0,C 180,E1 -25335.984,E2 -25335.984} C_VEL
LIN {X 0,Y 166.414,Z 453.745,A -85,B 0,C 180,E1 -25336.811,E2 -25336.811} C_VEL
LIN {X 0,Y 167.845,Z 443.374,A -85,B 0,C 180,E1 -25337.415,E2 -25337.415} C_VEL
LIN {X 0,Y 169.367,Z 424.151,A -85,B 0,C 180,E1 -25338.157,E2 -25338.157} C_VEL
LIN {X 0,Y 169.174,Z 420.351,A -85,B 0,C 180,E1 -25338.466,E2 -25338.466} C_VEL
LIN {X 0,Y 167.909,Z 415.753,A -85,B 0,C 180,E1 -25339.246,E2 -25339.246} C_VEL
LIN {X 0,Y 163.885,Z 406.094,A -85,B 0,C 180,E1 -25341.554,E2 -25341.554} C_VEL
LIN {X 0,Y 160.9,Z 398.214,A -85,B 0,C 180,E1 -25343.476,E2 -25343.476} C_VEL
LIN {X 0,Y 156.453,Z 387.989,A -85,B 0,C 180,E1 -25346.54,E2 -25346.54} C_VEL
LIN {X 0,Y 152.773,Z 380.814,A -85,B 0,C 180,E1 -25349.312,E2 -25349.312} C_VEL
LIN {X 0,Y 148.811,Z 374.721,A -85,B 0,C 180,E1 -25352.581,E2 -25352.581} C_VEL
LIN {X 0,Y 145.694,Z 370.392,A -85,B 0,C 180,E1 -25355.522,E2 -25355.522} C_VEL
LIN {X 0,Y 142.822,Z 366.6,A -85,B 0,C 180,E1 -25358.666,E2 -25358.666} C_VEL
LIN {X 0,Y 141.958,Z 365.513,A -85,B 0,C 180,E1 -25359.722,E2 -25359.722} C_VEL
LIN {X 0,Y 139.422,Z 362.445,A -85,B 0,C 180,E1 -25363.25,E2 -25363.25} C_VEL
LIN {X 0,Y 138.587,Z 360.73,A -85,B 0,C 180,E1 -25364.746,E2 -25364.746} C_VEL
LIN {X 0,Y 135.885,Z 358.398,A -85,B 0,C 180,E1 -25370.306,E2 -25370.306} C_VEL
LIN {X 0,Y 134.655,Z 355.647,A -85,B 0,C 180,E1 -25375.508,E2 -25375.508} C_VEL
LIN {X 0,Y 134.306,Z 354.835,A -85,B 0,C 180,E1 -25379.998,E2 -25379.998} C_VEL
LIN {X 0,Y 134.707,Z 355.811,A -85,B 0,C 180,E1 -25385.237,E2 -25385.237} C_VEL
LIN {X 0,Y 137.488,Z 360.121,A -85,B 0,C 180,E1 -25393.75,E2 -25393.75} C_VEL
LIN {X 0,Y 138.783,Z 361.017,A -85,B 0,C 180,E1 -25395.982,E2 -25395.982} C_VEL
LIN {X 0,Y 140.626,Z 364.217,A -85,B 0,C 180,E1 -25398.955,E2 -25398.955} C_VEL
LIN {X 0,Y 142.727,Z 366.384,A -85,B 0,C 180,E1 -25401.592,E2 -25401.592} C_VEL
LIN {X 0,Y 145.291,Z 369.979,A -85,B 0,C 180,E1 -25404.466,E2 -25404.466} C_VEL
LIN {X 0,Y 146.519,Z 371.584,A -85,B 0,C 180,E1 -25405.689,E2 -25405.689} C_VEL
LIN {X 0,Y 149.775,Z 376.246,A -85,B 0,C 180,E1 -25408.651,E2 -25408.651} C_VEL
LIN {X 0,Y 154.269,Z 382.897,A -85,B 0,C 180,E1 -25412.17,E2 -25412.17} C_VEL
LIN {X 0,Y 159.682,Z 392.071,A -85,B 0,C 180,E1 -25415.856,E2 -25415.856} C_VEL
LIN {X 0,Y 164.691,Z 401.776,A -85,B 0,C 180,E1 -25418.886,E2 -25418.886} C_VEL
LIN {X 0,Y 168.911,Z 411.169,A -85,B 0,C 180,E1 -25421.239,E2 -25421.239} C_VEL
LIN {X 0,Y 174.159,Z 425.076,A -85,B 0,C 180,E1 -25424.002,E2 -25424.002} C_VEL
LIN {X 0,Y 180.439,Z 440.003,A -85,B 0,C 180,E1 -25427.012,E2 -25427.012} C_VEL
LIN {X 0,Y 185.983,Z 451.873,A -85,B 0,C 180,E1 -25429.841,E2 -25429.841} C_VEL
LIN {X 0,Y 191.731,Z 462.726,A -85,B 0,C 180,E1 -25432.807,E2 -25432.807} C_VEL
LIN {X 0,Y 197.743,Z 472.167,A -85,B 0,C 180,E1 -25435.721,E2 -25435.721} C_VEL
LIN {X 0,Y 205.267,Z 482.07,A -85,B 0,C 180,E1 -25439.099,E2 -25439.099} C_VEL
LIN {X 0,Y 214.093,Z 491.529,A -85,B 0,C 180,E1 -25442.641,E2 -25442.641} C_VEL
LIN {X 0,Y 223.333,Z 499.353,A -85,B 0,C 180,E1 -25445.863,E2 -25445.863} C_VEL
LIN {X 0,Y 236.081,Z 507.813,A -85,B 0,C 180,E1 -25449.672,E2 -25449.672} C_VEL
LIN {X 0,Y 249.561,Z 515.146,A -85,B 0,C 180,E1 -25453.23,E2 -25453.23} C_VEL
LIN {X 0,Y 260.682,Z 520.629,A -85,B 0,C 180,E1 -25456.059,E2 -25456.059} C_VEL
LIN {X 0,Y 267.431,Z 523.933,A -85,B 0,C 180,E1 -25457.864,E2 -25457.864} C_VEL
LIN {X 0,Y 273.456,Z 526.964,A -85,B 0,C 180,E1 -25459.636,E2 -25459.636} C_VEL
LIN {X 0,Y 278.657,Z 529.56,A -85,B 0,C 180,E1 -25461.296,E2 -25461.296} C_VEL
LIN {X 0,Y 283.098,Z 532.141,A -85,B 0,C 180,E1 -25463.215,E2 -25463.215} C_VEL
LIN {X 0,Y 285.288,Z 533.419,A -85,B 0,C 180,E1 -25464.345,E2 -25464.345} C_VEL
LIN {X 0,Y 288.728,Z 535.167,A -85,B 0,C 180,E1 -25466.354,E2 -25466.354} C_VEL
LIN {X 0,Y 289.848,Z 535.648,A -85,B 0,C 180,E1 -25467.22,E2 -25467.22} C_VEL
LIN {X 0,Y 291.108,Z 536.154,A -85,B 0,C 180,E1 -25468.617,E2 -25468.617} C_VEL
LIN {X 0,Y 291.779,Z 536.299,A -85,B 0,C 180,E1 -25470,E2 -25470} C_VEL
LIN {X 0,Y 291.142,Z 536.155,A -85,B 0,C 180,E1 -25471.383,E2 -25471.383} C_VEL
LIN {X 0,Y 289.86,Z 535.648,A -85,B 0,C 180,E1 -25472.779,E2 -25472.779} C_VEL
LIN {X 0,Y 287.818,Z 534.734,A -85,B 0,C 180,E1 -25474.201,E2 -25474.201} C_VEL
LIN {X 0,Y 285.284,Z 533.419,A -85,B 0,C 180,E1 -25475.655,E2 -25475.655} C_VEL
LIN {X 0,Y 282.317,Z 531.708,A -85,B 0,C 180,E1 -25477.15,E2 -25477.15} C_VEL
LIN {X 0,Y 278.679,Z 529.559,A -85,B 0,C 180,E1 -25478.703,E2 -25478.703} C_VEL
LIN {X 0,Y 271.912,Z 526.178,A -85,B 0,C 180,E1 -25480.841,E2 -25480.841} C_VEL
LIN {X 0,Y 263.493,Z 521.943,A -85,B 0,C 180,E1 -25483.214,E2 -25483.214} C_VEL
LIN {X 0,Y 251.771,Z 516.224,A -85,B 0,C 180,E1 -25486.209,E2 -25486.209} C_VEL
LIN {X 0,Y 238.728,Z 509.348,A -85,B 0,C 180,E1 -25489.603,E2 -25489.603} C_VEL
LIN {X 0,Y 225.823,Z 501.159,A -85,B 0,C 180,E1 -25493.354,E2 -25493.354} C_VEL
LIN {X 0,Y 216.171,Z 493.379,A -85,B 0,C 180,E1 -25496.616,E2 -25496.616} C_VEL
LIN {X 0,Y 208.263,Z 485.487,A -85,B 0,C 180,E1 -25499.666,E2 -25499.666} C_VEL
LIN {X 0,Y 199.765,Z 475.069,A -85,B 0,C 180,E1 -25503.328,E2 -25503.328} C_VEL
LIN {X 0,Y 193.744,Z 466.09,A -85,B 0,C 180,E1 -25506.187,E2 -25506.187} C_VEL
LIN {X 0,Y 188.908,Z 457.657,A -85,B 0,C 180,E1 -25508.625,E2 -25508.625} C_VEL
LIN {X 0,Y 183.535,Z 446.871,A -85,B 0,C 180,E1 -25511.386,E2 -25511.386} C_VEL
LIN {X 0,Y 178.58,Z 435.795,A -85,B 0,C 180,E1 -25513.891,E2 -25513.891} C_VEL
LIN {X 0,Y 172.275,Z 419.968,A -85,B 0,C 180,E1 -25516.961,E2 -25516.961} C_VEL
LIN {X 0,Y 167.527,Z 407.88,A -85,B 0,C 180,E1 -25519.521,E2 -25519.521} C_VEL
LIN {X 0,Y 162.413,Z 397.162,A -85,B 0,C 180,E1 -25522.457,E2 -25522.457} C_VEL
LIN {X 0,Y 157.128,Z 387.653,A -85,B 0,C 180,E1 -25525.815,E2 -25525.815} C_VEL
LIN {X 0,Y 153.095,Z 381.17,A -85,B 0,C 180,E1 -25528.695,E2 -25528.695} C_VEL
LIN {X 0,Y 148.619,Z 374.474,A -85,B 0,C 180,E1 -25532.364,E2 -25532.364} C_VEL
LIN {X 0,Y 145.618,Z 370.301,A -85,B 0,C 180,E1 -25535.212,E2 -25535.212} C_VEL
LIN {X 0,Y 142.915,Z 366.742,A -85,B 0,C 180,E1 -25538.169,E2 -25538.169} C_VEL
LIN {X 0,Y 142.234,Z 365.744,A -85,B 0,C 180,E1 -25539.01,E2 -25539.01} C_VEL
LIN {X 0,Y 139.607,Z 362.773,A -85,B 0,C 180,E1 -25542.563,E2 -25542.563} C_VEL
LIN {X 0,Y 138.689,Z 360.803,A -85,B 0,C 180,E1 -25544.196,E2 -25544.196} C_VEL
LIN {X 0,Y 136.015,Z 358.602,A -85,B 0,C 180,E1 -25549.554,E2 -25549.554} C_VEL
LIN {X 0,Y 134.594,Z 355.568,A -85,B 0,C 180,E1 -25555.509,E2 -25555.509} C_VEL
LIN {X 0,Y 134.304,Z 354.855,A -85,B 0,C 180,E1 -25560.002,E2 -25560.002} C_VEL
LIN {X 0,Y 134.71,Z 355.811,A -85,B 0,C 180,E1 -25564.865,E2 -25564.865} C_VEL
LIN {X 0,Y 137.455,Z 360.091,A -85,B 0,C 180,E1 -25573.304,E2 -25573.304} C_VEL
LIN {X 0,Y 138.741,Z 360.926,A -85,B 0,C 180,E1 -25575.519,E2 -25575.519} C_VEL
LIN {X 0,Y 140.665,Z 364.248,A -85,B 0,C 180,E1 -25578.622,E2 -25578.622} C_VEL
LIN {X 0,Y 142.728,Z 366.415,A -85,B 0,C 180,E1 -25581.212,E2 -25581.212} C_VEL
LIN {X 0,Y 145.461,Z 370.142,A -85,B 0,C 180,E1 -25584.249,E2 -25584.249} C_VEL
LIN {X 0,Y 146.751,Z 371.94,A -85,B 0,C 180,E1 -25585.534,E2 -25585.534} C_VEL
LIN {X 0,Y 149.689,Z 376.134,A -85,B 0,C 180,E1 -25588.195,E2 -25588.195} C_VEL
LIN {X 0,Y 153.172,Z 381.32,A -85,B 0,C 180,E1 -25590.982,E2 -25590.982} C_VEL
LIN {X 0,Y 157.08,Z 389.344,A -85,B 0,C 180,E1 -25593.91,E2 -25593.91} C_VEL
LIN {X 0,Y 162.399,Z 401.836,A -85,B 0,C 180,E1 -25597.484,E2 -25597.484} C_VEL
LIN {X 0,Y 165.631,Z 411.126,A -85,B 0,C 180,E1 -25599.531,E2 -25599.531} C_VEL
LIN {X 0,Y 163.079,Z 443.495,A -85,B 0,C 180,E1 -25600.748,E2 -25600.748} C_VEL
LIN {X 0,Y 161.182,Z 456.305,A -85,B 0,C 180,E1 -25601.541,E2 -25601.541} C_VEL
LIN {X 0,Y 158,Z 469.653,A -85,B 0,C 180,E1 -25602.784,E2 -25602.784} C_VEL
LIN {X 0,Y 155.081,Z 479.162,A -85,B 0,C 180,E1 -25603.994,E2 -25603.994} C_VEL
LIN {X 0,Y 151.695,Z 488.432,A -85,B 0,C 180,E1 -25605.515,E2 -25605.515} C_VEL
LIN {X 0,Y 147.924,Z 497.37,A -85,B 0,C 180,E1 -25607.389,E2 -25607.389} C_VEL
LIN {X 0,Y 143.802,Z 505.892,A -85,B 0,C 180,E1 -25609.643,E2 -25609.643} C_VEL
LIN {X 0,Y 139.979,Z 513.107,A -85,B 0,C 180,E1 -25612.046,E2 -25612.046} C_VEL
LIN {X 0,Y 136.424,Z 519.305,A -85,B 0,C 180,E1 -25614.582,E2 -25614.582} C_VEL
LIN {X 0,Y 132.439,Z 525.841,A -85,B 0,C 180,E1 -25617.951,E2 -25617.951} C_VEL
LIN {X 0,Y 129.757,Z 530.348,A -85,B 0,C 180,E1 -25620.827,E2 -25620.827} C_VEL
LIN {X 0,Y 126.001,Z 535.838,A -85,B 0,C 180,E1 -25625.271,E2 -25625.271} C_VEL
LIN {X 0,Y 123.006,Z 540.163,A -85,B 0,C 180,E1 -25629.952,E2 -25629.952} C_VEL
LIN {X 0,Y 121.604,Z 542.536,A -85,B 0,C 180,E1 -25633.204,E2 -25633.204} C_VEL
LIN {X 0,Y 120.525,Z 544.341,A -85,B 0,C 180,E1 -25636.512,E2 -25636.512} C_VEL
LIN {X 0,Y 119.392,Z 546.803,A -85,B 0,C 180,E1 -25643.239,E2 -25643.239} C_VEL
LIN {X 0,Y 119.231,Z 547.398,A -85,B 0,C 180,E1 -25646.621,E2 -25646.621} C_VEL
LIN {X 0,Y 119.337,Z 547.559,A -85,B 0,C 180,E1 -25650,E2 -25650} C_VEL
LIN {X 0,Y 119.222,Z 547.398,A -85,B 0,C 180,E1 -25653.379,E2 -25653.379} C_VEL
LIN {X 0,Y 119.331,Z 546.801,A -85,B 0,C 180,E1 -25656.764,E2 -25656.764} C_VEL
LIN {X 0,Y 120.524,Z 544.341,A -85,B 0,C 180,E1 -25663.488,E2 -25663.488} C_VEL
LIN {X 0,Y 122.245,Z 541.382,A -85,B 0,C 180,E1 -25668.433,E2 -25668.433} C_VEL
LIN {X 0,Y 124.915,Z 537.392,A -85,B 0,C 180,E1 -25673.193,E2 -25673.193} C_VEL
LIN {X 0,Y 128.391,Z 532.262,A -85,B 0,C 180,E1 -25677.728,E2 -25677.728} C_VEL
LIN {X 0,Y 132.147,Z 526.416,A -85,B 0,C 180,E1 -25681.684,E2 -25681.684} C_VEL
LIN {X 0,Y 135.588,Z 520.681,A -85,B 0,C 180,E1 -25684.761,E2 -25684.761} C_VEL
LIN {X 0,Y 139.075,Z 514.733,A -85,B 0,C 180,E1 -25687.329,E2 -25687.329} C_VEL
LIN {X 0,Y 142.83,Z 507.811,A -85,B 0,C 180,E1 -25689.766,E2 -25689.766} C_VEL
LIN {X 0,Y 146.853,Z 499.637,A -85,B 0,C 180,E1 -25692.066,E2 -25692.066} C_VEL
LIN {X 0,Y 150.585,Z 491.133,A -85,B 0,C 180,E1 -25693.965,E2 -25693.965} C_VEL
LIN {X 0,Y 153.906,Z 482.422,A -85,B 0,C 180,E1 -25695.519,E2 -25695.519} C_VEL
LIN {X 0,Y 157.084,Z 472.671,A -85,B 0,C 180,E1 -25696.871,E2 -25696.871} C_VEL
LIN {X 0,Y 159.457,Z 463.883,A -85,B 0,C 180,E1 -25697.815,E2 -25697.815} C_VEL
LIN {X 0,Y 161.703,Z 453.11,A -85,B 0,C 180,E1 -25698.679,E2 -25698.679} C_VEL
LIN {X 0,Y 163.123,Z 443.181,A -85,B 0,C 180,E1 -25699.252,E2 -25699.252} C_VEL
LIN {X 0,Y 165.626,Z 411.183,A -85,B 0,C 180,E1 -25700.467,E2 -25700.467} C_VEL
LIN {X 0,Y 163.885,Z 406.094,A -85,B 0,C 180,E1 -25701.554,E2 -25701.554} C_VEL
LIN {X 0,Y 162.623,Z 403.099,A -85,B 0,C 180,E1 -25702.324,E2 -25702.324} C_VEL
LIN {X 0,Y 161.034,Z 400.592,A -85,B 0,C 180,E1 -25703.239,E2 -25703.239} C_VEL
LIN {X 0,Y 157.412,Z 396.562,A -85,B 0,C 180,E1 -25705.343,E2 -25705.343} C_VEL
LIN {X 0,Y 153.799,Z 392.817,A -85,B 0,C 180,E1 -25707.643,E2 -25707.643} C_VEL
LIN {X 0,Y 151.526,Z 389.436,A -85,B 0,C 180,E1 -25709.32,E2 -25709.32} C_VEL
LIN {X 0,Y 150.906,Z 388.097,A -85,B 0,C 180,E1 -25709.839,E2 -25709.839} C_VEL
LIN {X 0,Y 148.166,Z 383.48,A -85,B 0,C 180,E1 -25712.164,E2 -25712.164} C_VEL
LIN {X 0,Y 145.944,Z 380.091,A -85,B 0,C 180,E1 -25714.219,E2 -25714.219} C_VEL
LIN {X 0,Y 143.342,Z 376.342,A -85,B 0,C 180,E1 -25716.905,E2 -25716.905} C_VEL
LIN {X 0,Y 140.431,Z 372.205,A -85,B 0,C 180,E1 -25720.445,E2 -25720.445} C_VEL
LIN {X 0,Y 137.907,Z 368.992,A -85,B 0,C 180,E1 -25724.196,E2 -25724.196} C_VEL
LIN {X 0,Y 137.209,Z 367.531,A -85,B 0,C 180,E1 -25725.538,E2 -25725.538} C_VEL
LIN {X 0,Y 134.761,Z 365.224,A -85,B 0,C 180,E1 -25730.997,E2 -25730.997} C_VEL
LIN {X 0,Y 133.678,Z 362.542,A -85,B 0,C 180,E1 -25736.23,E2 -25736.23} C_VEL
LIN {X 0,Y 133.442,Z 361.873,A -85,B 0,C 180,E1 -25739.998,E2 -25739.998} C_VEL
LIN {X 0,Y 133.775,Z 362.822,A -85,B 0,C 180,E1 -25744.896,E2 -25744.896} C_VEL
LIN {X 0,Y 136.232,Z 366.934,A -85,B 0,C 180,E1 -25753.043,E2 -25753.043} C_VEL
LIN {X 0,Y 137.392,Z 367.842,A -85,B 0,C 180,E1 -25755.196,E2 -25755.196} C_VEL
LIN {X 0,Y 139.612,Z 371.457,A -85,B 0,C 180,E1 -25758.863,E2 -25758.863} C_VEL
LIN {X 0,Y 141.045,Z 372.995,A -85,B 0,C 180,E1 -25760.735,E2 -25760.735} C_VEL
LIN {X 0,Y 143.491,Z 376.527,A -85,B 0,C 180,E1 -25763.64,E2 -25763.64} C_VEL
LIN {X 0,Y 147.314,Z 382.139,A -85,B 0,C 180,E1 -25767.452,E2 -25767.452} C_VEL
LIN {X 0,Y 151.499,Z 388.603,A -85,B 0,C 180,E1 -25770.972,E2 -25770.972} C_VEL
LIN {X 0,Y 156.579,Z 397.647,A -85,B 0,C 180,E1 -25774.687,E2 -25774.687} C_VEL
LIN {X 0,Y 161.125,Z 406.782,A -85,B 0,C 180,E1 -25777.635,E2 -25777.635} C_VEL
LIN {X 0,Y 165.236,Z 416.467,A -85,B 0,C 180,E1 -25780.106,E2 -25780.106} C_VEL
LIN {X 0,Y 172.69,Z 436.663,A -85,B 0,C 180,E1 -25784.282,E2 -25784.282} C_VEL
LIN {X 0,Y 176.323,Z 445.739,A -85,B 0,C 180,E1 -25786.357,E2 -25786.357} C_VEL
LIN {X 0,Y 180.116,Z 454.488,A -85,B 0,C 180,E1 -25788.6,E2 -25788.6} C_VEL
LIN {X 0,Y 184.861,Z 464.17,A -85,B 0,C 180,E1 -25791.387,E2 -25791.387} C_VEL
LIN {X 0,Y 190.235,Z 473.392,A -85,B 0,C 180,E1 -25794.365,E2 -25794.365} C_VEL
LIN {X 0,Y 196.449,Z 482.343,A -85,B 0,C 180,E1 -25797.546,E2 -25797.546} C_VEL
LIN {X 0,Y 203.404,Z 490.635,A -85,B 0,C 180,E1 -25800.764,E2 -25800.764} C_VEL
LIN {X 0,Y 211.204,Z 498.18,A -85,B 0,C 180,E1 -25803.952,E2 -25803.952} C_VEL
LIN {X 0,Y 221.823,Z 506.171,A -85,B 0,C 180,E1 -25807.655,E2 -25807.655} C_VEL
LIN {X 0,Y 233.824,Z 513.244,A -85,B 0,C 180,E1 -25811.222,E2 -25811.222} C_VEL
LIN {X 0,Y 247.536,Z 519.912,A -85,B 0,C 180,E1 -25814.863,E2 -25814.863} C_VEL
LIN {X 0,Y 258.834,Z 524.94,A -85,B 0,C 180,E1 -25817.816,E2 -25817.816} C_VEL
LIN {X 0,Y 267.137,Z 528.71,A -85,B 0,C 180,E1 -25820.234,E2 -25820.234} C_VEL
LIN {X 0,Y 270.234,Z 530.09,A -85,B 0,C 180,E1 -25821.208,E2 -25821.208} C_VEL
LIN {X 0,Y 274.145,Z 531.933,A -85,B 0,C 180,E1 -25822.636,E2 -25822.636} C_VEL
LIN {X 0,Y 277.396,Z 533.637,A -85,B 0,C 180,E1 -25824.184,E2 -25824.184} C_VEL
LIN {X 0,Y 281.62,Z 535.555,A -85,B 0,C 180,E1 -25826.569,E2 -25826.569} C_VEL
LIN {X 0,Y 282.43,Z 535.87,A -85,B 0,C 180,E1 -25827.147,E2 -25827.147} C_VEL
LIN {X 0,Y 283.876,Z 536.428,A -85,B 0,C 180,E1 -25828.581,E2 -25828.581} C_VEL
LIN {X 0,Y 284.646,Z 536.611,A -85,B 0,C 180,E1 -25830,E2 -25830} C_VEL
LIN {X 0,Y 283.903,Z 536.426,A -85,B 0,C 180,E1 -25831.418,E2 -25831.418} C_VEL
LIN {X 0,Y 282.437,Z 535.87,A -85,B 0,C 180,E1 -25832.853,E2 -25832.853} C_VEL
LIN {X 0,Y 280.102,Z 534.943,A -85,B 0,C 180,E1 -25834.317,E2 -25834.317} C_VEL
LIN {X 0,Y 275.899,Z 532.846,A -85,B 0,C 180,E1 -25836.57,E2 -25836.57} C_VEL
LIN {X 0,Y 274.159,Z 531.933,A -85,B 0,C 180,E1 -25837.364,E2 -25837.364} C_VEL
LIN {X 0,Y 269.628,Z 529.809,A -85,B 0,C 180,E1 -25838.997,E2 -25838.997} C_VEL
LIN {X 0,Y 261.343,Z 526.095,A -85,B 0,C 180,E1 -25841.477,E2 -25841.477} C_VEL
LIN {X 0,Y 253.151,Z 522.434,A -85,B 0,C 180,E1 -25843.675,E2 -25843.675} C_VEL
LIN {X 0,Y 241.977,Z 517.315,A -85,B 0,C 180,E1 -25846.577,E2 -25846.577} C_VEL
LIN {X 0,Y 228.732,Z 510.436,A -85,B 0,C 180,E1 -25850.227,E2 -25850.227} C_VEL
LIN {X 0,Y 215.958,Z 502.018,A -85,B 0,C 180,E1 -25854.329,E2 -25854.329} C_VEL
LIN {X 0,Y 205.455,Z 492.792,A -85,B 0,C 180,E1 -25858.362,E2 -25858.362} C_VEL
LIN {X 0,Y 197,Z 483.084,A -85,B 0,C 180,E1 -25862.18,E2 -25862.18} C_VEL
LIN {X 0,Y 191.367,Z 475.215,A -85,B 0,C 180,E1 -25865.022,E2 -25865.022} C_VEL
LIN {X 0,Y 186.494,Z 467.179,A -85,B 0,C 180,E1 -25867.687,E2 -25867.687} C_VEL
LIN {X 0,Y 182.003,Z 458.438,A -85,B 0,C 180,E1 -25870.305,E2 -25870.305} C_VEL
LIN {X 0,Y 177.457,Z 448.37,A -85,B 0,C 180,E1 -25872.995,E2 -25872.995} C_VEL
LIN {X 0,Y 172.959,Z 437.307,A -85,B 0,C 180,E1 -25875.602,E2 -25875.602} C_VEL
LIN {X 0,Y 164.705,Z 415.11,A -85,B 0,C 180,E1 -25880.206,E2 -25880.206} C_VEL
LIN {X 0,Y 160.68,Z 405.825,A -85,B 0,C 180,E1 -25882.642,E2 -25882.642} C_VEL
LIN {X 0,Y 156.082,Z 396.743,A -85,B 0,C 180,E1 -25885.652,E2 -25885.652} C_VEL
LIN {X 0,Y 151.31,Z 388.264,A -85,B 0,C 180,E1 -25889.18,E2 -25889.18} C_VEL
LIN {X 0,Y 146.365,Z 380.673,A -85,B 0,C 180,E1 -25893.436,E2 -25893.436} C_VEL
LIN {X 0,Y 143.647,Z 376.697,A -85,B 0,C 180,E1 -25896.196,E2 -25896.196} C_VEL
LIN {X 0,Y 140.899,Z 372.754,A -85,B 0,C 180,E1 -25899.458,E2 -25899.458} C_VEL
LIN {X 0,Y 138.002,Z 369.179,A -85,B 0,C 180,E1 -25903.641,E2 -25903.641} C_VEL
LIN {X 0,Y 137.2,Z 367.565,A -85,B 0,C 180,E1 -25905.162,E2 -25905.162} C_VEL
LIN {X 0,Y 134.819,Z 365.297,A -85,B 0,C 180,E1 -25910.439,E2 -25910.439} C_VEL
LIN {X 0,Y 133.628,Z 362.469,A -85,B 0,C 180,E1 -25916.232,E2 -25916.232} C_VEL
LIN {X 0,Y 133.441,Z 361.883,A -85,B 0,C 180,E1 -25920.002,E2 -25920.002} C_VEL
LIN {X 0,Y 133.776,Z 362.828,A -85,B 0,C 180,E1 -25924.521,E2 -25924.521} C_VEL
LIN {X 0,Y 136.416,Z 367.083,A -85,B 0,C 180,E1 -25933.028,E2 -25933.028} C_VEL
LIN {X 0,Y 137.398,Z 367.835,A -85,B 0,C 180,E1 -25934.82,E2 -25934.82} C_VEL
LIN {X 0,Y 139.401,Z 371.188,A -85,B 0,C 180,E1 -25938.178,E2 -25938.178} C_VEL
LIN {X 0,Y 141.084,Z 373.107,A -85,B 0,C 180,E1 -25940.409,E2 -25940.409} C_VEL
LIN {X 0,Y 144.574,Z 378.069,A -85,B 0,C 180,E1 -25944.408,E2 -25944.408} C_VEL
LIN {X 0,Y 147.551,Z 382.547,A -85,B 0,C 180,E1 -25947.289,E2 -25947.289} C_VEL
LIN {X 0,Y 150.395,Z 386.991,A -85,B 0,C 180,E1 -25949.723,E2 -25949.723} C_VEL
LIN {X 0,Y 154.274,Z 395.392,A -85,B 0,C 180,E1 -25952.848,E2 -25952.848} C_VEL
LIN {X 0,Y 159.09,Z 407.577,A -85,B 0,C 180,E1 -25956.342,E2 -25956.342} C_VEL
LIN {X 0,Y 161.011,Z 413.376,A -85,B 0,C 180,E1 -25957.67,E2 -25957.67} C_VEL
LIN {X 0,Y 158.537,Z 443.308,A -85,B 0,C 180,E1 -25958.805,E2 -25958.805} C_VEL
LIN {X 0,Y 156.467,Z 456.644,A -85,B 0,C 180,E1 -25959.632,E2 -25959.632} C_VEL
LIN {X 0,Y 153.275,Z 469.459,A -85,B 0,C 180,E1 -25960.84,E2 -25960.84} C_VEL
LIN {X 0,Y 150.237,Z 478.968,A -85,B 0,C 180,E1 -25962.046,E2 -25962.046} C_VEL
LIN {X 0,Y 146.709,Z 488.238,A -85,B 0,C 180,E1 -25963.57,E2 -25963.57} C_VEL
LIN {X 0,Y 142.763,Z 497.176,A -85,B 0,C 180,E1 -25965.453,E2 -25965.453} C_VEL
LIN {X 0,Y 138.447,Z 505.698,A -85,B 0,C 180,E1 -25967.732,E2 -25967.732} C_VEL
LIN {X 0,Y 134.446,Z 512.913,A -85,B 0,C 180,E1 -25970.183,E2 -25970.183} C_VEL
LIN {X 0,Y 130.686,Z 519.111,A -85,B 0,C 180,E1 -25972.772,E2 -25972.772} C_VEL
LIN {X 0,Y 126.44,Z 525.646,A -85,B 0,C 180,E1 -25976.233,E2 -25976.233} C_VEL
LIN {X 0,Y 123.56,Z 530.152,A -85,B 0,C 180,E1 -25979.209,E2 -25979.209} C_VEL
LIN {X 0,Y 119.552,Z 535.643,A -85,B 0,C 180,E1 -25983.84,E2 -25983.84} C_VEL
LIN {X 0,Y 116.341,Z 539.969,A -85,B 0,C 180,E1 -25988.75,E2 -25988.75} C_VEL
LIN {X 0,Y 114.773,Z 542.341,A -85,B 0,C 180,E1 -25992.172,E2 -25992.172} C_VEL
LIN {X 0,Y 113.616,Z 544.147,A -85,B 0,C 180,E1 -25995.675,E2 -25995.675} C_VEL
LIN {X 0,Y 112.316,Z 546.608,A -85,B 0,C 180,E1 -26002.811,E2 -26002.811} C_VEL
LIN {X 0,Y 112.139,Z 547.204,A -85,B 0,C 180,E1 -26006.407,E2 -26006.407} C_VEL
LIN {X 0,Y 112.253,Z 547.366,A -85,B 0,C 180,E1 -26010,E2 -26010} C_VEL
LIN {X 0,Y 112.129,Z 547.204,A -85,B 0,C 180,E1 -26013.593,E2 -26013.593} C_VEL
LIN {X 0,Y 112.267,Z 546.607,A -85,B 0,C 180,E1 -26017.192,E2 -26017.192} C_VEL
LIN {X 0,Y 113.615,Z 544.147,A -85,B 0,C 180,E1 -26024.325,E2 -26024.325} C_VEL
LIN {X 0,Y 115.496,Z 541.187,A -85,B 0,C 180,E1 -26029.553,E2 -26029.553} C_VEL
LIN {X 0,Y 118.405,Z 537.197,A -85,B 0,C 180,E1 -26034.549,E2 -26034.549} C_VEL
LIN {X 0,Y 122.141,Z 532.068,A -85,B 0,C 180,E1 -26039.28,E2 -26039.28} C_VEL
LIN {X 0,Y 125.737,Z 526.802,A -85,B 0,C 180,E1 -26043.023,E2 -26043.023} C_VEL
LIN {X 0,Y 129.802,Z 520.486,A -85,B 0,C 180,E1 -26046.553,E2 -26046.553} C_VEL
LIN {X 0,Y 133.477,Z 514.539,A -85,B 0,C 180,E1 -26049.185,E2 -26049.185} C_VEL
LIN {X 0,Y 137.431,Z 507.616,A -85,B 0,C 180,E1 -26051.666,E2 -26051.666} C_VEL
LIN {X 0,Y 141.653,Z 499.443,A -85,B 0,C 180,E1 -26053.994,E2 -26053.994} C_VEL
LIN {X 0,Y 145.559,Z 490.939,A -85,B 0,C 180,E1 -26055.905,E2 -26055.905} C_VEL
LIN {X 0,Y 149.018,Z 482.229,A -85,B 0,C 180,E1 -26057.467,E2 -26057.467} C_VEL
LIN {X 0,Y 152.332,Z 472.478,A -85,B 0,C 180,E1 -26058.814,E2 -26058.814} C_VEL
LIN {X 0,Y 154.776,Z 463.689,A -85,B 0,C 180,E1 -26059.764,E2 -26059.764} C_VEL
LIN {X 0,Y 157.007,Z 453.505,A -85,B 0,C 180,E1 -26060.583,E2 -26060.583} C_VEL
LIN {X 0,Y 158.534,Z 443.431,A -85,B 0,C 180,E1 -26061.174,E2 -26061.174} C_VEL
LIN {X 0,Y 161.003,Z 413.465,A -85,B 0,C 180,E1 -26062.328,E2 -26062.328} C_VEL
LIN {X 0,Y 157.521,Z 403.365,A -85,B 0,C 180,E1 -26064.759,E2 -26064.759} C_VEL
LIN {X 0,Y 153.031,Z 392.559,A -85,B 0,C 180,E1 -26068.118,E2 -26068.118} C_VEL
LIN {X 0,Y 150.906,Z 388.097,A -85,B 0,C 180,E1 -26069.839,E2 -26069.839} C_VEL
LIN {X 0,Y 149.609,Z 385.774,A -85,B 0,C 180,E1 -26070.921,E2 -26070.921} C_VEL
LIN {X 0,Y 148.085,Z 384.14,A -85,B 0,C 180,E1 -26072.156,E2 -26072.156} C_VEL
LIN {X 0,Y 144.823,Z 382.289,A -85,B 0,C 180,E1 -26074.895,E2 -26074.895} C_VEL
LIN {X 0,Y 140.276,Z 380.32,A -85,B 0,C 180,E1 -26079.441,E2 -26079.441} C_VEL
LIN {X 0,Y 139.084,Z 379.09,A -85,B 0,C 180,E1 -26080.966,E2 -26080.966} C_VEL
LIN {X 0,Y 136.475,Z 375.618,A -85,B 0,C 180,E1 -26085.078,E2 -26085.078} C_VEL
LIN {X 0,Y 135.955,Z 374.415,A -85,B 0,C 180,E1 -26086.166,E2 -26086.166} C_VEL
LIN {X 0,Y 133.558,Z 371.866,A -85,B 0,C 180,E1 -26092.059,E2 -26092.059} C_VEL
LIN {X 0,Y 132.722,Z 369.444,A -85,B 0,C 180,E1 -26096.963,E2 -26096.963} C_VEL
LIN {X 0,Y 132.574,Z 368.939,A -85,B 0,C 180,E1 -26099.998,E2 -26099.998} C_VEL
LIN {X 0,Y 132.806,Z 369.648,A -85,B 0,C 180,E1 -26104.171,E2 -26104.171} C_VEL
LIN {X 0,Y 135.2,Z 373.936,A -85,B 0,C 180,E1 -26112.762,E2 -26112.762} C_VEL
LIN {X 0,Y 136.098,Z 374.767,A -85,B 0,C 180,E1 -26114.531,E2 -26114.531} C_VEL
LIN {X 0,Y 138.29,Z 378.33,A -85,B 0,C 180,E1 -26118.328,E2 -26118.328} C_VEL
LIN {X 0,Y 139.448,Z 379.76,A -85,B 0,C 180,E1 -26119.943,E2 -26119.943} C_VEL
LIN {X 0,Y 142.524,Z 384.35,A -85,B 0,C 180,E1 -26123.714,E2 -26123.714} C_VEL
LIN {X 0,Y 145.228,Z 388.563,A -85,B 0,C 180,E1 -26126.52,E2 -26126.52} C_VEL
LIN {X 0,Y 148.797,Z 394.31,A -85,B 0,C 180,E1 -26129.73,E2 -26129.73} C_VEL
LIN {X 0,Y 153.49,Z 403.048,A -85,B 0,C 180,E1 -26133.426,E2 -26133.426} C_VEL
